C05476=1016.184,128.856,379.831,166.835,54.880,160.081
C05477=1016.188,129.105,379.813,166.839,54.870,160.080
C05478=1016.193,129.355,379.795,166.841,54.860,160.079
C05479=1016.197,129.605,379.776,166.845,54.850,160.077
C05480=1016.202,129.853,379.757,166.848,54.840,160.076
C05481=1016.207,130.103,379.739,166.851,54.831,160.075
C05482=1016.211,130.352,379.720,166.854,54.820,160.073
C05483=1016.216,130.601,379.702,166.858,54.811,160.072
C05484=1016.220,130.851,379.683,166.860,54.801,160.071
C05485=1016.225,131.099,379.664,166.863,54.791,160.069
C05486=1016.231,131.349,379.645,166.867,54.781,160.068
C05487=1016.235,131.598,379.626,166.869,54.771,160.067
C05488=1016.240,131.848,379.608,166.873,54.761,160.066
C05489=1016.244,132.097,379.589,166.876,54.751,160.065
C05490=1016.249,132.346,379.570,166.879,54.741,160.063
C05491=1016.254,132.596,379.552,166.882,54.731,160.062
C05492=1016.258,132.845,379.533,166.886,54.721,160.061
C05493=1016.263,133.094,379.514,166.888,54.712,160.059
C05494=1016.267,133.343,379.495,166.891,54.701,160.058
C05495=1016.272,133.592,379.477,166.895,54.692,160.057
C05496=1016.277,133.841,379.458,166.898,54.681,160.055
C05497=1016.282,134.091,379.439,166.901,54.672,160.054
C05498=1016.287,134.340,379.420,166.904,54.662,160.053
C05499=1016.291,134.590,379.401,166.908,54.652,160.052
C05500=1016.296,134.839,379.382,166.910,54.642,160.050
C05501=1016.301,135.088,379.364,166.914,54.632,160.049
C05502=1016.305,135.337,379.345,166.917,54.622,160.048
C05503=1016.310,135.586,379.326,166.921,54.612,160.046
C05504=1016.314,135.835,379.307,166.923,54.602,160.045
C05505=1016.320,136.085,379.288,166.927,54.592,160.044
C05506=1016.324,136.334,379.269,166.930,54.582,160.043
C05507=1016.329,136.583,379.250,166.932,54.572,160.041
C05508=1016.333,136.833,379.231,166.936,54.563,160.040
C05509=1016.338,137.082,379.212,166.939,54.552,160.039
C05510=1016.342,137.331,379.194,166.943,54.542,160.037
C05511=1016.348,137.581,379.174,166.946,54.533,160.036
C05512=1016.352,137.830,379.155,166.949,54.523,160.035
C05513=1016.357,138.079,379.137,166.952,54.512,160.034
C05514=1016.361,138.328,379.117,166.955,54.503,160.032
C05515=1016.366,138.609,379.095,166.959,54.492,160.031
C05516=1016.372,138.890,379.074,166.963,54.481,160.030
C05517=1016.377,139.171,379.053,166.966,54.470,160.028
C05518=1016.382,139.452,379.031,166.970,54.458,160.027
C05519=1016.387,139.702,379.011,166.974,54.449,160.026
C05520=1016.392,139.951,378.993,166.977,54.439,160.024
C05521=1016.396,140.200,378.973,166.980,54.429,160.023
C05522=1016.400,140.449,378.954,166.983,54.419,160.022
C05523=1016.406,140.699,378.935,166.986,54.409,160.020
C05524=1016.410,140.948,378.915,166.989,54.400,160.019
C05525=1016.415,141.197,378.896,166.993,54.390,160.018
C05526=1016.420,141.446,378.878,166.996,54.379,160.017
C05527=1016.424,141.695,378.858,167.000,54.370,160.016
C05528=1016.429,141.945,378.838,167.002,54.360,160.014
C05529=1016.434,142.194,378.819,167.006,54.350,160.013
C05530=1016.438,142.443,378.800,167.010,54.340,160.012
C05531=1016.442,142.692,378.781,167.013,54.330,160.010
C05532=1016.448,142.942,378.762,167.015,54.320,160.009
C05533=1016.452,143.191,378.742,167.019,54.311,160.008
C05534=1016.457,143.440,378.723,167.023,54.301,160.007
C05535=1016.462,143.689,378.704,167.026,54.290,160.005
C05536=1016.467,143.938,378.684,167.029,54.281,160.004
C05537=1016.471,144.187,378.665,167.032,54.271,160.003
C05538=1016.476,144.436,378.646,167.036,54.261,160.001
C05539=1016.481,144.686,378.626,167.040,54.251,160.000
C05540=1016.485,144.935,378.607,167.043,54.241,159.999
C05541=1016.490,145.184,378.588,167.045,54.231,159.998
C05542=1016.495,145.434,378.569,167.049,54.222,159.997
C05543=1016.500,145.683,378.549,167.053,54.212,159.995
C05544=1016.504,145.932,378.530,167.056,54.202,159.994
C05545=1016.509,146.182,378.510,167.059,54.192,159.993
C05546=1016.514,146.430,378.491,167.062,54.182,159.991
C05547=1016.518,146.680,378.472,167.066,54.173,159.990
C05548=1016.523,146.928,378.451,167.070,54.163,159.989
C05549=1016.528,147.178,378.431,167.072,54.153,159.988
C05550=1016.532,147.427,378.412,167.076,54.143,159.987
C05551=1016.537,147.676,378.392,167.080,54.133,159.985
C05552=1016.542,147.926,378.373,167.083,54.124,159.984
C05553=1016.546,148.175,378.353,167.086,54.114,159.983
C05554=1016.552,148.424,378.334,167.089,54.104,159.982
C05555=1016.556,148.673,378.315,167.093,54.094,159.980
C05556=1016.560,148.922,378.295,167.097,54.084,159.979
C05557=1016.566,149.171,378.274,167.100,54.075,159.978
C05558=1016.570,149.420,378.255,167.103,54.065,159.977
C05559=1016.574,149.669,378.236,167.107,54.055,159.975
C05560=1016.579,149.919,378.216,167.110,54.045,159.974
C05561=1016.584,150.168,378.196,167.113,54.035,159.973
C05562=1016.589,150.418,378.176,167.117,54.026,159.972
C05563=1016.593,150.666,378.156,167.120,54.016,159.971
C05564=1016.598,150.915,378.137,167.124,54.006,159.969
C05565=1016.602,151.165,378.117,167.128,53.996,159.968
C05566=1016.607,151.414,378.097,167.130,53.986,159.967
C05567=1016.612,151.663,378.077,167.134,53.977,159.966
C05568=1016.616,151.912,378.057,167.138,53.967,159.964
C05569=1016.621,152.161,378.038,167.141,53.957,159.963
C05570=1016.626,152.411,378.018,167.145,53.947,159.962
C05571=1016.630,152.659,377.998,167.148,53.938,159.961
C05572=1016.635,152.909,377.978,167.152,53.928,159.960
C05573=1016.640,153.158,377.959,167.155,53.918,159.958
C05574=1016.645,153.407,377.938,167.159,53.908,159.957
C05575=1016.649,153.656,377.919,167.162,53.898,159.956
C05576=1016.654,153.906,377.899,167.165,53.889,159.954
C05577=1016.659,154.155,377.879,167.169,53.879,159.953
C05578=1016.663,154.404,377.859,167.172,53.869,159.952
C05579=1016.668,154.685,377.835,167.177,53.858,159.951
C05580=1016.674,154.966,377.814,167.181,53.847,159.950
C05581=1016.679,155.247,377.791,167.184,53.837,159.948
C05582=1016.685,155.528,377.769,167.188,53.825,159.947
C05583=1016.689,155.778,377.748,167.192,53.815,159.945
C05584=1016.693,156.026,377.728,167.196,53.806,159.944
C05585=1016.698,156.276,377.708,167.199,53.796,159.943
C05586=1016.703,156.524,377.688,167.203,53.786,159.942
C05587=1016.708,156.774,377.668,167.206,53.777,159.941
C05588=1016.713,157.022,377.648,167.210,53.767,159.940
C05589=1016.718,157.272,377.628,167.213,53.757,159.938
C05590=1016.722,157.521,377.608,167.217,53.747,159.937
C05591=1016.727,157.770,377.588,167.221,53.738,159.936
C05592=1016.731,158.019,377.567,167.224,53.727,159.935
C05593=1016.736,158.269,377.547,167.227,53.718,159.933
C05594=1016.741,158.517,377.527,167.231,53.708,159.932
C05595=1016.746,158.767,377.507,167.235,53.699,159.931
C05596=1016.750,159.016,377.487,167.238,53.689,159.930
C05597=1016.754,159.265,377.465,167.241,53.680,159.929
C05598=1016.759,159.514,377.445,167.245,53.670,159.928
C05599=1016.763,159.764,377.425,167.249,53.660,159.926
C05600=1016.768,160.012,377.405,167.253,53.651,159.925
C05601=1016.772,160.261,377.383,167.256,53.642,159.924
C05602=1016.777,160.511,377.363,167.260,53.632,159.923
C05603=1016.781,160.759,377.342,167.264,53.623,159.922
C05604=1016.785,161.009,377.322,167.268,53.613,159.921
C05605=1016.790,161.258,377.302,167.270,53.603,159.919
C05606=1016.795,161.507,377.280,167.274,53.594,159.918
C05607=1016.799,161.756,377.260,167.278,53.584,159.917
C05608=1016.804,162.005,377.239,167.282,53.575,159.916
C05609=1016.808,162.255,377.218,167.285,53.566,159.915
C05610=1016.813,162.504,377.198,167.288,53.556,159.913
C05611=1016.817,162.753,377.177,167.292,53.546,159.912
C05612=1016.822,163.001,377.157,167.297,53.537,159.911
C05613=1016.826,163.251,377.136,167.299,53.527,159.910
C05614=1016.832,163.500,377.115,167.303,53.518,159.909
C05615=1016.836,163.749,377.095,167.307,53.508,159.908
C05616=1016.840,163.998,377.073,167.311,53.498,159.906
C05617=1016.845,164.247,377.053,167.315,53.489,159.905
C05618=1016.849,164.496,377.032,167.317,53.479,159.904
C05619=1016.855,164.745,377.012,167.321,53.470,159.903
C05620=1016.858,164.994,376.991,167.325,53.460,159.902
C05621=1016.863,165.244,376.970,167.329,53.451,159.901
C05622=1016.868,165.493,376.950,167.333,53.441,159.900
C05623=1016.872,165.742,376.929,167.337,53.431,159.898
C05624=1016.877,165.991,376.908,167.340,53.422,159.897
C05625=1016.882,166.240,376.887,167.343,53.412,159.896
C05626=1016.885,166.489,376.867,167.348,53.403,159.895
C05627=1016.891,166.738,376.846,167.352,53.394,159.894
C05628=1016.895,166.988,376.825,167.355,53.384,159.892
C05629=1016.900,167.236,376.805,167.359,53.374,159.891
C05630=1016.904,167.486,376.783,167.362,53.365,159.890
C05631=1016.909,167.735,376.762,167.366,53.355,159.889
C05632=1016.914,167.984,376.742,167.370,53.346,159.888
C05633=1016.918,168.233,376.721,167.374,53.336,159.887
C05634=1016.923,168.482,376.700,167.378,53.327,159.886
C05635=1016.928,168.731,376.679,167.381,53.317,159.884
C05636=1016.932,168.979,376.658,167.386,53.307,159.883
C05637=1016.937,169.229,376.637,167.390,53.298,159.882
C05638=1016.942,169.478,376.616,167.393,53.288,159.881
C05639=1016.947,169.727,376.596,167.396,53.279,159.880
C05640=1016.951,169.976,376.575,167.400,53.269,159.878
C05641=1016.956,170.225,376.554,167.404,53.260,159.877
C05642=1016.961,170.474,376.533,167.408,53.250,159.876
C05643=1016.966,170.755,376.509,167.412,53.239,159.875
C05644=1016.971,171.036,376.485,167.417,53.228,159.874
C05645=1016.977,171.317,376.462,167.421,53.218,159.872
C05646=1016.983,171.597,376.438,167.426,53.207,159.871
C05647=1016.986,171.846,376.417,167.429,53.197,159.870
C05648=1016.992,172.095,376.397,167.433,53.187,159.869
C05649=1016.996,172.345,376.376,167.438,53.178,159.868
C05650=1017.001,172.594,376.354,167.441,53.168,159.866
C05651=1017.006,172.843,376.334,167.445,53.159,159.865
C05652=1017.011,173.092,376.312,167.449,53.149,159.864
C05653=1017.015,173.340,376.292,167.453,53.140,159.863
C05654=1017.020,173.590,376.271,167.457,53.130,159.862
C05655=1017.024,173.839,376.250,167.461,53.120,159.861
C05656=1017.030,174.088,376.228,167.465,53.110,159.859
C05657=1017.035,174.337,376.207,167.469,53.101,159.858
C05658=1017.039,174.587,376.186,167.473,53.092,159.857
C05659=1017.044,174.836,376.165,167.477,53.082,159.856
C05660=1017.049,175.084,376.144,167.481,53.073,159.855
C05661=1017.054,175.333,376.123,167.484,53.063,159.854
C05662=1017.058,175.582,376.102,167.489,53.053,159.853
C05663=1017.063,175.831,376.080,167.492,53.043,159.851
C05664=1017.068,176.080,376.060,167.496,53.034,159.850
C05665=1017.073,176.330,376.039,167.500,53.024,159.849
C05666=1017.078,176.579,376.018,167.504,53.015,159.848
C05667=1017.083,176.828,375.996,167.508,53.006,159.847
C05668=1017.088,177.077,375.975,167.512,52.996,159.846
C05669=1017.093,177.326,375.954,167.516,52.986,159.845
C05670=1017.098,177.575,375.933,167.520,52.976,159.843
C05671=1017.102,177.825,375.912,167.524,52.967,159.842
C05672=1017.108,178.073,375.890,167.528,52.957,159.841
C05673=1017.112,178.323,375.869,167.532,52.948,159.840
C05674=1017.117,178.571,375.849,167.536,52.938,159.839
C05675=1017.122,178.820,375.827,167.540,52.929,159.838
C05676=1017.126,179.069,375.806,167.544,52.919,159.837
C05677=1017.132,179.318,375.785,167.548,52.910,159.835
C05678=1017.136,179.567,375.764,167.553,52.899,159.834
C05679=1017.141,179.816,375.742,167.557,52.890,159.833
C05680=1017.146,180.065,375.721,167.561,52.881,159.832
C05681=1017.151,180.315,375.700,167.565,52.871,159.831
C05682=1017.156,180.563,375.679,167.569,52.862,159.830
C05683=1017.161,180.812,375.658,167.573,52.852,159.829
C05684=1017.166,181.062,375.635,167.577,52.843,159.828
C05685=1017.172,181.311,375.615,167.581,52.833,159.826
C05686=1017.176,181.560,375.593,167.585,52.823,159.825
C05687=1017.181,181.809,375.572,167.590,52.813,159.824
C05688=1017.186,182.058,375.550,167.594,52.804,159.823
C05689=1017.191,182.307,375.528,167.597,52.795,159.822
C05690=1017.195,182.556,375.506,167.601,52.786,159.821
C05691=1017.199,182.806,375.484,167.605,52.777,159.820
C05692=1017.204,183.054,375.463,167.610,52.767,159.819
C05693=1017.209,183.303,375.441,167.614,52.758,159.818
C05694=1017.213,183.552,375.418,167.618,52.749,159.817
C05695=1017.218,183.801,375.396,167.622,52.739,159.815
C05696=1017.223,184.050,375.375,167.626,52.730,159.814
C05697=1017.227,184.299,375.353,167.630,52.721,159.813
C05698=1017.232,184.548,375.330,167.635,52.711,159.812
C05699=1017.236,184.797,375.308,167.639,52.702,159.811
C05700=1017.241,185.045,375.286,167.643,52.693,159.810
C05701=1017.245,185.295,375.265,167.647,52.684,159.809
C05702=1017.250,185.544,375.243,167.651,52.675,159.808
C05703=1017.255,185.794,375.221,167.655,52.665,159.807
C05704=1017.260,186.042,375.199,167.659,52.656,159.806
C05705=1017.264,186.292,375.176,167.664,52.646,159.805
C05706=1017.269,186.540,375.154,167.668,52.637,159.804
C05707=1017.275,186.820,375.129,167.673,52.627,159.803
C05708=1017.280,187.101,375.104,167.677,52.616,159.801
C05709=1017.285,187.381,375.080,167.682,52.606,159.800
C05710=1017.290,187.662,375.055,167.687,52.596,159.799
C05711=1017.294,187.910,375.033,167.691,52.586,159.798
C05712=1017.300,188.160,375.011,167.695,52.577,159.797
C05713=1017.304,188.409,374.988,167.699,52.568,159.796
C05714=1017.309,188.658,374.966,167.703,52.558,159.795
C05715=1017.314,188.906,374.944,167.708,52.549,159.794
C05716=1017.319,189.155,374.922,167.712,52.540,159.792
C05717=1017.323,189.404,374.900,167.716,52.531,159.791
C05718=1017.328,189.654,374.877,167.721,52.521,159.791
C05719=1017.333,189.902,374.855,167.726,52.512,159.789
C05720=1017.337,190.152,374.833,167.730,52.503,159.788
C05721=1017.342,190.400,374.811,167.734,52.494,159.787
C05722=1017.347,190.649,374.789,167.738,52.484,159.786
C05723=1017.352,190.899,374.767,167.742,52.475,159.785
C05724=1017.357,191.147,374.744,167.746,52.465,159.784
C05725=1017.361,191.396,374.722,167.751,52.456,159.783
C05726=1017.366,191.645,374.700,167.755,52.447,159.782
C05727=1017.371,191.895,374.677,167.759,52.438,159.781
C05728=1017.376,192.143,374.655,167.765,52.429,159.780
C05729=1017.381,192.392,374.633,167.769,52.419,159.779
C05730=1017.386,192.640,374.611,167.773,52.410,159.778
C05731=1017.390,192.890,374.588,167.777,52.400,159.777
C05732=1017.395,193.139,374.566,167.781,52.391,159.776
C05733=1017.400,193.387,374.544,167.786,52.382,159.775
C05734=1017.405,193.637,374.521,167.790,52.373,159.774
C05735=1017.410,193.886,374.499,167.795,52.364,159.773
C05736=1017.415,194.135,374.477,167.799,52.354,159.772
C05737=1017.419,194.383,374.454,167.804,52.345,159.771
C05738=1017.424,194.633,374.432,167.808,52.335,159.769
C05739=1017.429,194.882,374.410,167.812,52.326,159.768
C05740=1017.434,195.130,374.387,167.816,52.317,159.767
C05741=1017.439,195.380,374.364,167.822,52.308,159.766
C05742=1017.444,195.628,374.343,167.826,52.299,159.765
C05743=1017.450,195.877,374.320,167.830,52.289,159.764
C05744=1017.454,196.126,374.297,167.834,52.280,159.763
C05745=1017.459,196.375,374.275,167.839,52.271,159.762
C05746=1017.464,196.624,374.252,167.844,52.262,159.761
C05747=1017.468,196.873,374.230,167.848,52.253,159.760
C05748=1017.474,197.121,374.207,167.852,52.243,159.759
C05749=1017.479,197.371,374.185,167.857,52.234,159.758
C05750=1017.483,197.620,374.163,167.862,52.224,159.757
C05751=1017.489,197.869,374.140,167.866,52.215,159.756
C05752=1017.494,198.118,374.118,167.871,52.206,159.755
C05753=1017.499,198.367,374.095,167.875,52.197,159.754
C05754=1017.503,198.616,374.072,167.880,52.188,159.753
C05755=1017.509,198.864,374.050,167.885,52.178,159.752
C05756=1017.514,199.114,374.028,167.889,52.169,159.751
C05757=1017.518,199.362,374.004,167.893,52.160,159.750
C05758=1017.523,199.612,373.982,167.899,52.151,159.749
C05759=1017.528,199.860,373.959,167.903,52.142,159.748
C05760=1017.533,200.109,373.936,167.907,52.133,159.747
C05761=1017.537,200.358,373.913,167.912,52.124,159.746
C05762=1017.543,200.607,373.890,167.916,52.114,159.745
C05763=1017.547,200.856,373.867,167.920,52.105,159.744
C05764=1017.552,201.104,373.844,167.926,52.096,159.743
C05765=1017.557,201.354,373.822,167.930,52.087,159.742
C05766=1017.562,201.602,373.798,167.935,52.078,159.741
C05767=1017.567,201.852,373.775,167.939,52.069,159.740
C05768=1017.572,202.100,373.752,167.943,52.060,159.739
C05769=1017.577,202.349,373.729,167.949,52.051,159.738
C05770=1017.600,203.593,373.613,168.432,52.137,159.849
C05771=1017.606,203.828,373.591,168.436,52.129,159.848
C05772=1017.612,204.063,373.567,168.440,52.122,159.847
C05773=1017.618,204.298,373.544,168.443,52.114,159.846
C05774=1017.623,204.534,373.521,168.447,52.107,159.845
C05775=1017.629,204.769,373.498,168.450,52.099,159.844
C05776=1017.634,205.003,373.474,168.454,52.091,159.844
C05777=1017.640,205.238,373.451,168.458,52.084,159.843
C05778=1017.645,205.473,373.428,168.462,52.076,159.842
C05779=1017.651,205.722,373.402,168.466,52.068,159.841
C05780=1017.657,205.970,373.378,168.470,52.061,159.840
C05781=1017.663,206.219,373.353,168.474,52.053,159.839
C05782=1017.669,206.468,373.328,168.477,52.045,159.838
C05783=1017.674,206.716,373.303,168.481,52.037,159.837
C05784=1017.680,206.966,373.279,168.485,52.030,159.836
C05785=1017.686,207.214,373.254,168.490,52.021,159.835
C05786=1017.692,207.463,373.229,168.494,52.013,159.834
C05787=1017.698,207.712,373.204,168.498,52.006,159.834
C05788=1017.703,207.960,373.179,168.501,51.998,159.833
C05789=1017.709,208.209,373.154,168.505,51.990,159.832
C05790=1017.716,208.458,373.129,168.509,51.983,159.831
C05791=1017.721,208.706,373.104,168.513,51.975,159.830
C05792=1017.727,208.955,373.079,168.517,51.967,159.829
C05793=1017.732,209.204,373.054,168.521,51.960,159.828
C05794=1017.738,209.452,373.029,168.525,51.951,159.827
C05795=1017.744,209.701,373.004,168.530,51.944,159.826
C05796=1017.750,209.950,372.978,168.533,51.936,159.825
C05797=1017.756,210.198,372.954,168.537,51.929,159.825
C05798=1017.762,210.447,372.929,168.541,51.921,159.824
C05799=1017.767,210.696,372.903,168.545,51.913,159.823
C05800=1017.773,210.944,372.878,168.549,51.905,159.822
C05801=1017.779,211.193,372.853,168.553,51.898,159.821
C05802=1017.785,211.442,372.828,168.557,51.890,159.820
C05803=1017.790,211.690,372.802,168.561,51.883,159.819
C05804=1017.796,211.939,372.777,168.565,51.876,159.818
C05805=1017.802,212.187,372.752,168.569,51.868,159.817
C05806=1017.808,212.436,372.726,168.573,51.860,159.817
C05807=1017.813,212.685,372.701,168.577,51.853,159.816
C05808=1017.819,212.934,372.676,168.581,51.845,159.815
C05809=1017.825,213.182,372.651,168.585,51.838,159.814
C05810=1017.831,213.431,372.625,168.589,51.830,159.813
C05811=1017.836,213.679,372.600,168.593,51.823,159.812
C05812=1017.843,213.928,372.574,168.597,51.816,159.811
C05813=1017.849,214.177,372.549,168.601,51.808,159.810
C05814=1017.854,214.426,372.523,168.605,51.800,159.810
C05815=1017.860,214.674,372.499,168.609,51.793,159.809
C05816=1017.866,214.923,372.474,168.613,51.786,159.808
C05817=1017.871,215.172,372.448,168.617,51.778,159.807
C05818=1017.878,215.421,372.422,168.621,51.771,159.806
C05819=1017.884,215.669,372.397,168.625,51.763,159.806
C05820=1017.889,215.917,372.372,168.630,51.756,159.805
C05821=1017.895,216.166,372.346,168.633,51.748,159.804
C05822=1017.901,216.415,372.321,168.636,51.741,159.803
C05823=1017.907,216.663,372.295,168.641,51.734,159.802
C05824=1017.913,216.912,372.270,168.645,51.727,159.801
C05825=1017.919,217.161,372.244,168.648,51.719,159.800
C05826=1017.925,217.410,372.219,168.653,51.712,159.799
C05827=1017.931,217.658,372.194,168.657,51.704,159.799
C05828=1017.937,217.906,372.168,168.661,51.697,159.798
C05829=1017.943,218.155,372.142,168.665,51.690,159.797
C05830=1017.949,218.403,372.116,168.669,51.683,159.796
C05831=1017.959,218.817,372.074,168.675,51.671,159.795
C05832=1017.966,219.179,372.036,168.681,51.660,159.794
C05833=1017.975,219.540,371.998,168.687,51.650,159.793
C05834=1017.983,219.901,371.961,168.693,51.640,159.792
C05835=1017.992,220.263,371.923,168.699,51.629,159.790
C05836=1017.998,220.512,371.897,168.704,51.622,159.790
C05837=1018.003,220.760,371.872,168.708,51.615,159.789
C05838=1018.009,221.009,371.846,168.712,51.608,159.788
C05839=1018.015,221.257,371.820,168.716,51.600,159.787
C05840=1018.021,221.506,371.794,168.719,51.594,159.786
C05841=1018.026,221.755,371.768,168.723,51.586,159.786
C05842=1018.033,222.003,371.742,168.728,51.580,159.785
C05843=1018.038,222.252,371.716,168.732,51.573,159.784
C05844=1018.044,222.500,371.691,168.736,51.565,159.783
C05845=1018.050,222.749,371.664,168.741,51.558,159.783
C05846=1018.056,222.997,371.639,168.744,51.551,159.782
C05847=1018.062,223.246,371.613,168.748,51.544,159.781
C05848=1018.068,223.495,371.587,168.753,51.537,159.780
C05849=1018.074,223.743,371.561,168.757,51.530,159.780
C05850=1018.080,223.992,371.535,168.761,51.523,159.779
C05851=1018.086,224.240,371.509,168.765,51.516,159.778
C05852=1018.091,224.489,371.483,168.769,51.510,159.777
C05853=1018.097,224.738,371.457,168.773,51.502,159.777
C05854=1018.103,224.986,371.431,168.777,51.495,159.776
C05855=1018.109,225.235,371.405,168.781,51.488,159.775
C05856=1018.115,225.483,371.379,168.786,51.482,159.774
C05857=1018.121,225.732,371.353,168.789,51.475,159.774
C05858=1018.127,225.980,371.327,168.793,51.467,159.773
C05859=1018.133,226.229,371.301,168.798,51.461,159.772
C05860=1018.138,226.478,371.275,168.802,51.454,159.771
C05861=1018.145,226.726,371.249,168.806,51.447,159.771
C05862=1018.151,226.974,371.222,168.810,51.440,159.770
C05863=1018.156,227.223,371.196,168.814,51.433,159.769
C05864=1018.162,227.471,371.169,168.819,51.427,159.769
C05865=1018.168,227.720,371.142,168.822,51.420,159.768
C05866=1018.174,227.969,371.117,168.827,51.413,159.767
C05867=1018.180,228.218,371.090,168.831,51.406,159.766
C05868=1018.186,228.466,371.064,168.836,51.400,159.766
C05869=1018.191,228.715,371.038,168.839,51.393,159.765
C05870=1018.197,228.963,371.011,168.843,51.386,159.764
C05871=1018.203,229.212,370.985,168.848,51.379,159.764
C05872=1018.209,229.460,370.958,168.851,51.373,159.763
C05873=1018.215,229.709,370.933,168.856,51.366,159.762
C05874=1018.221,229.957,370.906,168.860,51.359,159.762
C05875=1018.227,230.205,370.879,168.865,51.353,159.761
C05876=1018.233,230.454,370.852,168.868,51.347,159.760
C05877=1018.239,230.703,370.826,168.873,51.339,159.759
C05878=1018.244,230.951,370.799,168.877,51.333,159.759
C05879=1018.250,231.199,370.772,168.881,51.327,159.758
C05880=1018.256,231.448,370.746,168.885,51.320,159.757
C05881=1018.262,231.697,370.720,168.890,51.313,159.757
C05882=1018.267,231.945,370.693,168.893,51.307,159.756
C05883=1018.274,232.194,370.666,168.898,51.300,159.755
C05884=1018.279,232.443,370.639,168.902,51.293,159.755
C05885=1018.285,232.691,370.613,168.906,51.287,159.754
C05886=1018.291,232.939,370.586,168.911,51.281,159.754
C05887=1018.297,233.188,370.559,168.914,51.275,159.753
C05888=1018.302,233.416,370.535,168.919,51.268,159.752
C05889=1018.308,233.644,370.510,168.922,51.262,159.752
C05890=1018.313,233.872,370.486,168.926,51.256,159.751
C05891=1018.318,234.101,370.461,168.930,51.250,159.750
C05892=1018.324,234.329,370.437,168.934,51.244,159.750
C05893=1018.330,234.558,370.412,168.937,51.238,159.749
C05894=1018.334,234.786,370.387,168.941,51.233,159.749
C05895=1018.341,235.014,370.363,168.945,51.226,159.748
C05896=1018.346,235.262,370.337,168.950,51.220,159.747
C05897=1018.353,235.511,370.310,168.954,51.213,159.747
C05898=1018.358,235.760,370.283,168.958,51.207,159.746
C05899=1018.365,236.007,370.256,168.963,51.201,159.746
C05900=1018.370,236.256,370.229,168.966,51.195,159.745
C05901=1018.377,236.505,370.202,168.971,51.188,159.744
C05902=1018.382,236.753,370.175,168.976,51.182,159.744
C05903=1018.387,237.002,370.148,168.979,51.176,159.743
C05904=1018.393,237.250,370.121,168.984,51.169,159.743
C05905=1018.400,237.499,370.094,168.988,51.162,159.742
C05906=1018.406,237.747,370.067,168.992,51.156,159.741
C05907=1018.412,237.995,370.040,168.997,51.150,159.741
C05908=1018.418,238.244,370.013,169.000,51.144,159.740
C05909=1018.424,238.493,369.987,169.005,51.138,159.739
C05910=1018.429,238.741,369.960,169.010,51.131,159.739
C05911=1018.436,238.990,369.932,169.013,51.125,159.738
C05912=1018.442,239.238,369.906,169.018,51.118,159.738
C05913=1018.447,239.487,369.878,169.022,51.112,159.737
C05914=1018.454,239.735,369.851,169.026,51.106,159.736
C05915=1018.459,239.983,369.824,169.030,51.100,159.736
C05916=1018.465,240.231,369.796,169.035,51.094,159.735
C05917=1018.471,240.481,369.769,169.039,51.088,159.735
C05918=1018.477,240.729,369.742,169.043,51.081,159.734
C05919=1018.483,240.978,369.714,169.047,51.075,159.733
C05920=1018.489,241.226,369.687,169.052,51.070,159.733
C05921=1018.495,241.474,369.660,169.056,51.063,159.732
C05922=1018.500,241.723,369.632,169.061,51.057,159.732
C05923=1018.506,241.971,369.605,169.064,51.051,159.731
C05924=1018.513,242.220,369.578,169.069,51.045,159.731
C05925=1018.518,242.468,369.550,169.074,51.039,159.730
C05926=1018.524,242.716,369.523,169.078,51.033,159.729
C05927=1018.531,242.965,369.496,169.083,51.027,159.729
C05928=1018.536,243.213,369.468,169.086,51.021,159.728
C05929=1018.542,243.462,369.441,169.091,51.015,159.728
C05930=1018.548,243.710,369.413,169.095,51.009,159.727
C05931=1018.553,243.958,369.385,169.099,51.003,159.727
C05932=1018.559,244.207,369.358,169.104,50.997,159.726
C05933=1018.565,244.455,369.330,169.107,50.991,159.726
C05934=1018.571,244.704,369.302,169.113,50.985,159.725
C05935=1018.576,244.952,369.275,169.117,50.980,159.725
C05936=1018.582,245.201,369.247,169.121,50.973,159.724
C05937=1018.588,245.449,369.219,169.125,50.968,159.724
C05938=1018.594,245.697,369.191,169.130,50.961,159.723
C05939=1018.600,245.945,369.163,169.134,50.956,159.723
C05940=1018.606,246.195,369.136,169.138,50.950,159.722
C05941=1018.611,246.443,369.108,169.143,50.944,159.722
C05942=1018.617,246.691,369.080,169.147,50.939,159.721
C05943=1018.623,246.939,369.052,169.152,50.932,159.720
C05944=1018.629,247.188,369.024,169.156,50.927,159.720
C05945=1018.635,247.436,368.997,169.160,50.920,159.719
C05946=1018.641,247.685,368.969,169.164,50.915,159.719
C05947=1018.646,247.933,368.941,169.169,50.910,159.718
C05948=1018.652,248.158,368.915,169.173,50.904,159.718
C05949=1018.657,248.383,368.891,169.177,50.899,159.718
C05950=1018.663,248.608,368.865,169.181,50.893,159.717
C05951=1018.668,248.833,368.840,169.185,50.888,159.717
C05952=1018.674,249.058,368.815,169.189,50.883,159.716
C05953=1018.679,249.283,368.790,169.192,50.878,159.716
C05954=1018.684,249.507,368.765,169.196,50.873,159.715
C05955=1018.689,249.733,368.738,169.201,50.867,159.715
C05956=1018.696,249.981,368.711,169.205,50.862,159.714
C05957=1018.701,250.229,368.683,169.210,50.856,159.714
C05958=1018.708,250.478,368.655,169.214,50.851,159.714
C05959=1018.714,250.726,368.627,169.218,50.844,159.713
C05960=1018.719,250.974,368.599,169.223,50.839,159.712
C05961=1018.726,251.223,368.571,169.228,50.833,159.712
C05962=1018.731,251.471,368.543,169.232,50.828,159.712
C05963=1018.737,251.720,368.515,169.236,50.822,159.711
C05964=1018.744,251.968,368.487,169.240,50.816,159.711
C05965=1018.749,252.216,368.459,169.245,50.811,159.710
C05966=1018.755,252.465,368.431,169.250,50.805,159.710
C05967=1018.762,252.713,368.403,169.254,50.799,159.709
C05968=1018.767,252.961,368.375,169.259,50.794,159.709
C05969=1018.773,253.210,368.347,169.263,50.788,159.708
C05970=1018.780,253.459,368.319,169.267,50.783,159.708
C05971=1018.786,253.706,368.290,169.272,50.777,159.707
C05972=1018.792,253.954,368.262,169.276,50.771,159.707
C05973=1018.798,254.203,368.234,169.281,50.765,159.706
C05974=1018.804,254.452,368.206,169.285,50.760,159.706
C05975=1018.810,254.700,368.178,169.290,50.754,159.706
C05976=1018.816,254.948,368.150,169.294,50.749,159.705
C05977=1018.823,255.197,368.121,169.298,50.744,159.705
C05978=1018.829,255.445,368.093,169.303,50.738,159.704
C05979=1018.835,255.693,368.065,169.307,50.732,159.704
C05980=1018.840,255.942,368.037,169.313,50.727,159.703
C05981=1018.847,256.190,368.009,169.317,50.721,159.703
C05982=1018.853,256.438,367.980,169.322,50.716,159.703
C05983=1018.859,256.687,367.952,169.326,50.710,159.702
C05984=1018.865,256.935,367.925,169.330,50.705,159.702
C05985=1018.872,257.183,367.896,169.335,50.699,159.701
C05986=1018.878,257.432,367.867,169.339,50.694,159.701
C05987=1018.884,257.680,367.839,169.344,50.688,159.700
C05988=1018.891,257.928,367.810,169.348,50.683,159.700
C05989=1018.896,258.177,367.782,169.352,50.677,159.699
C05990=1018.903,258.425,367.755,169.358,50.672,159.699
C05991=1018.909,258.673,367.726,169.362,50.667,159.699
C05992=1018.915,258.922,367.697,169.367,50.661,159.698
C05993=1018.922,259.170,367.669,169.371,50.656,159.698
C05994=1018.928,259.418,367.641,169.376,50.650,159.697
C05995=1018.934,259.667,367.612,169.380,50.645,159.697
C05996=1018.941,259.915,367.584,169.385,50.639,159.697
C05997=1018.946,260.162,367.555,169.390,50.634,159.696
C05998=1018.952,260.411,367.527,169.394,50.629,159.696
C05999=1018.958,260.659,367.498,169.398,50.624,159.695
C06000=1018.965,260.907,367.469,169.404,50.618,159.695
C06001=1018.971,261.156,367.440,169.408,50.613,159.695
C06002=1018.976,261.404,367.411,169.412,50.608,159.694
C06003=1018.982,261.653,367.382,169.417,50.603,159.694
C06004=1018.988,261.901,367.353,169.422,50.597,159.694
C06005=1018.995,262.149,367.324,169.426,50.593,159.693
C06006=1019.000,262.397,367.296,169.431,50.587,159.693
C06007=1019.007,262.645,367.267,169.436,50.582,159.693
C06008=1019.012,262.870,367.241,169.440,50.578,159.692
C06009=1019.018,263.094,367.215,169.444,50.573,159.692
C06010=1019.023,263.318,367.188,169.448,50.569,159.692
C06011=1019.028,263.542,367.163,169.453,50.564,159.691
C06012=1019.034,263.766,367.137,169.457,50.558,159.691
C06013=1019.040,263.990,367.110,169.460,50.554,159.691
C06014=1019.045,264.214,367.084,169.465,50.549,159.690
C06015=1019.051,264.439,367.058,169.469,50.545,159.690
C06016=1019.057,264.687,367.029,169.474,50.540,159.690
C06017=1019.063,264.936,367.000,169.478,50.535,159.689
C06018=1019.069,265.184,366.971,169.483,50.530,159.689
C06019=1019.076,265.432,366.942,169.488,50.525,159.689
C06020=1019.082,265.680,366.913,169.492,50.520,159.688
C06021=1019.087,265.928,366.883,169.496,50.515,159.688
C06022=1019.094,266.176,366.854,169.502,50.510,159.688
C06023=1019.100,266.425,366.825,169.506,50.505,159.687
C06024=1019.106,266.673,366.796,169.511,50.500,159.687
C06025=1019.112,266.921,366.766,169.516,50.495,159.687
C06026=1019.118,267.169,366.737,169.520,50.490,159.686
C06027=1019.124,267.417,366.708,169.525,50.485,159.686
C06028=1019.130,267.666,366.679,169.530,50.480,159.686
C06029=1019.136,267.914,366.650,169.535,50.475,159.686
C06030=1019.142,268.162,366.621,169.539,50.470,159.685
C06031=1019.149,268.410,366.591,169.543,50.465,159.685
C06032=1019.155,268.658,366.562,169.549,50.460,159.685
C06033=1019.161,268.906,366.532,169.553,50.455,159.685
C06034=1019.167,269.154,366.503,169.558,50.451,159.684
C06035=1019.173,269.403,366.474,169.563,50.445,159.684
C06036=1019.179,269.651,366.445,169.568,50.440,159.684
C06037=1019.186,269.899,366.414,169.572,50.436,159.683
C06038=1019.192,270.147,366.385,169.577,50.431,159.683
C06039=1019.197,270.396,366.356,169.582,50.426,159.683
C06040=1019.204,270.643,366.326,169.587,50.421,159.683
C06041=1019.209,270.892,366.296,169.591,50.417,159.682
C06042=1019.216,271.140,366.267,169.596,50.412,159.682
C06043=1019.222,271.387,366.237,169.601,50.407,159.682
C06044=1019.228,271.636,366.207,169.606,50.402,159.682
C06045=1019.235,271.885,366.178,169.610,50.398,159.681
C06046=1019.240,272.132,366.148,169.615,50.393,159.681
C06047=1019.247,272.381,366.119,169.620,50.388,159.681
C06048=1019.252,272.629,366.089,169.625,50.383,159.681
C06049=1019.259,272.877,366.059,169.629,50.379,159.680
C06050=1019.265,273.126,366.030,169.634,50.374,159.680
C06051=1019.271,273.373,366.000,169.639,50.369,159.680
C06052=1019.277,273.622,365.970,169.644,50.364,159.679
C06053=1019.284,273.869,365.941,169.648,50.360,159.679
C06054=1019.290,274.118,365.911,169.653,50.355,159.679
C06055=1019.296,274.366,365.881,169.659,50.351,159.679
C06056=1019.302,274.614,365.851,169.663,50.346,159.679
C06057=1019.308,274.862,365.821,169.668,50.341,159.678
C06058=1019.315,275.110,365.791,169.672,50.337,159.678
C06059=1019.321,275.358,365.762,169.678,50.332,159.678
C06060=1019.327,275.606,365.731,169.683,50.328,159.678
C06061=1019.334,275.855,365.702,169.687,50.323,159.678
C06062=1019.339,276.103,365.671,169.692,50.318,159.677
C06063=1019.346,276.350,365.642,169.697,50.313,159.677
C06064=1019.351,276.599,365.612,169.702,50.309,159.677
C06065=1019.359,276.847,365.582,169.707,50.305,159.677
C06066=1019.364,277.095,365.552,169.711,50.300,159.676
C06067=1019.370,277.343,365.521,169.717,50.295,159.676
C06068=1019.376,277.570,365.494,169.720,50.291,159.676
C06069=1019.382,277.796,365.467,169.725,50.287,159.676
C06070=1019.387,278.022,365.439,169.730,50.283,159.676
C06071=1019.393,278.249,365.411,169.734,50.279,159.676
C06072=1019.398,278.475,365.383,169.739,50.275,159.675
C06073=1019.404,278.701,365.356,169.744,50.271,159.675
C06074=1019.410,278.928,365.329,169.747,50.267,159.675
C06075=1019.415,279.154,365.301,169.752,50.263,159.675
C06076=1019.422,279.403,365.270,169.757,50.259,159.675
C06077=1019.428,279.650,365.240,169.761,50.254,159.675
C06078=1019.435,279.899,365.209,169.767,50.250,159.675
C06079=1019.440,280.147,365.180,169.772,50.245,159.674
C06080=1019.446,280.395,365.150,169.777,50.241,159.674
C06081=1019.452,280.643,365.119,169.781,50.237,159.674
C06082=1019.459,280.891,365.089,169.787,50.232,159.674
C06083=1019.465,281.139,365.058,169.792,50.228,159.674
C06084=1019.471,281.387,365.028,169.797,50.224,159.674
C06085=1019.477,281.636,364.997,169.801,50.220,159.673
C06086=1019.484,281.883,364.967,169.806,50.215,159.673
C06087=1019.491,282.131,364.936,169.812,50.211,159.673
C06088=1019.497,282.379,364.906,169.816,50.206,159.673
C06089=1019.502,282.627,364.875,169.821,50.202,159.673
C06090=1019.509,282.875,364.845,169.826,50.198,159.673
C06091=1019.515,283.123,364.815,169.832,50.193,159.673
C06092=1019.522,283.371,364.784,169.837,50.189,159.672
C06093=1019.528,283.620,364.753,169.842,50.185,159.672
C06094=1019.534,283.868,364.723,169.846,50.180,159.672
C06095=1019.541,284.115,364.692,169.852,50.176,159.672
C06096=1019.547,284.363,364.662,169.857,50.172,159.672
C06097=1019.554,284.612,364.631,169.861,50.168,159.672
C06098=1019.560,284.859,364.601,169.866,50.164,159.672
C06099=1019.566,285.107,364.569,169.871,50.160,159.672
C06100=1019.572,285.355,364.539,169.877,50.155,159.672
C06101=1019.578,285.604,364.508,169.882,50.151,159.671
C06102=1019.585,285.851,364.477,169.887,50.147,159.671
C06103=1019.591,286.099,364.447,169.891,50.143,159.671
C06104=1019.597,286.348,364.416,169.896,50.139,159.671
C06105=1019.604,286.595,364.385,169.902,50.134,159.671
C06106=1019.610,286.844,364.354,169.907,50.130,159.671
C06107=1019.616,287.091,364.323,169.912,50.126,159.671
C06108=1019.623,287.339,364.292,169.917,50.123,159.671
C06109=1019.629,287.587,364.261,169.923,50.118,159.671
C06110=1019.635,287.835,364.230,169.928,50.114,159.671
C06111=1019.642,288.083,364.199,169.933,50.110,159.671
C06112=1019.648,288.332,364.168,169.938,50.106,159.670
C06113=1019.654,288.579,364.137,169.943,50.102,159.670
C06114=1019.661,288.827,364.107,169.948,50.098,159.670
C06115=1019.667,289.075,364.075,169.953,50.094,159.670
C06116=1019.673,289.323,364.045,169.958,50.090,159.670
C06117=1019.680,289.571,364.013,169.963,50.086,159.670
C06118=1019.687,289.819,363.982,169.968,50.082,159.670
C06119=1019.693,290.067,363.952,169.974,50.078,159.670
C06120=1019.699,290.315,363.920,169.979,50.074,159.670
C06121=1019.705,290.563,363.888,169.984,50.070,159.670
C06122=1019.711,290.811,363.858,169.989,50.066,159.670
C06123=1019.718,291.058,363.826,169.994,50.062,159.670
C06124=1019.725,291.306,363.795,170.000,50.058,159.670
C06125=1019.731,291.554,363.763,170.005,50.054,159.670
C06126=1019.737,291.802,363.733,170.010,50.050,159.670
C06127=1019.743,292.050,363.701,170.015,50.046,159.670
C06128=1019.750,292.283,363.672,170.020,50.043,159.670
C06129=1019.755,292.516,363.642,170.025,50.039,159.670
C06130=1019.762,292.748,363.613,170.030,50.036,159.670
C06131=1019.767,292.981,363.583,170.035,50.032,159.670
C06132=1019.774,293.213,363.554,170.039,50.028,159.669
C06133=1019.779,293.446,363.524,170.044,50.025,159.670
C06134=1019.785,293.678,363.495,170.050,50.022,159.670
C06135=1019.791,293.910,363.464,170.054,50.018,159.670
C06136=1019.797,294.158,363.433,170.060,50.014,159.670
C06137=1019.803,294.406,363.401,170.065,50.010,159.670
C06138=1019.810,294.654,363.369,170.070,50.007,159.670
C06139=1019.816,294.902,363.337,170.075,50.003,159.670
C06140=1019.822,295.150,363.306,170.080,50.000,159.670
C06141=1019.828,295.398,363.274,170.086,49.996,159.670
C06142=1019.834,295.645,363.242,170.091,49.992,159.670
C06143=1019.841,295.893,363.210,170.096,49.988,159.670
C06144=1019.847,296.142,363.178,170.102,49.985,159.670
C06145=1019.854,296.389,363.147,170.106,49.981,159.670
C06146=1019.860,296.638,363.115,170.112,49.978,159.670
C06147=1019.866,296.884,363.083,170.118,49.974,159.670
C06148=1019.872,297.132,363.051,170.123,49.970,159.670
C06149=1019.878,297.381,363.019,170.128,49.967,159.670
C06150=1019.885,297.628,362.987,170.133,49.963,159.670
C06151=1019.891,297.876,362.955,170.138,49.960,159.670
C06152=1019.898,298.124,362.923,170.144,49.956,159.670
C06153=1019.904,298.372,362.890,170.150,49.952,159.670
C06154=1019.911,298.620,362.859,170.155,49.949,159.670
C06155=1019.917,298.868,362.827,170.160,49.946,159.670
C06156=1019.923,299.115,362.794,170.165,49.942,159.671
C06157=1019.930,299.363,362.763,170.170,49.938,159.670
C06158=1019.936,299.611,362.731,170.177,49.935,159.671
C06159=1019.943,299.859,362.699,170.182,49.931,159.671
C06160=1019.949,300.107,362.667,170.187,49.928,159.671
C06161=1019.956,300.354,362.634,170.192,49.924,159.671
C06162=1019.962,300.602,362.602,170.197,49.921,159.671
C06163=1019.968,300.850,362.570,170.204,49.917,159.671
C06164=1019.975,301.098,362.538,170.209,49.914,159.671
C06165=1019.981,301.346,362.505,170.214,49.911,159.671
C06166=1019.988,301.593,362.474,170.219,49.907,159.671
C06167=1019.994,301.841,362.441,170.225,49.903,159.671
C06168=1020.001,302.089,362.409,170.231,49.900,159.671
C06169=1020.007,302.337,362.377,170.236,49.896,159.672
C06170=1020.014,302.585,362.344,170.241,49.893,159.672
C06171=1020.021,302.833,362.313,170.247,49.890,159.672
C06172=1020.027,303.080,362.280,170.252,49.887,159.672
C06173=1020.034,303.328,362.248,170.258,49.883,159.672
C06174=1020.040,303.576,362.216,170.264,49.880,159.672
C06175=1020.047,303.823,362.183,170.268,49.876,159.672
C06176=1020.054,304.071,362.151,170.274,49.872,159.672
C06177=1020.060,304.320,362.118,170.280,49.869,159.672
C06178=1020.067,304.567,362.086,170.285,49.866,159.672
C06179=1020.073,304.814,362.054,170.291,49.862,159.673
C06180=1020.080,305.062,362.021,170.296,49.859,159.673
C06181=1020.087,305.309,361.989,170.302,49.855,159.673
C06182=1020.093,305.558,361.956,170.308,49.853,159.673
C06183=1020.100,305.806,361.924,170.313,49.849,159.673
C06184=1020.107,306.053,361.891,170.318,49.846,159.673
C06185=1020.113,306.301,361.859,170.325,49.843,159.674
C06186=1020.121,306.549,361.826,170.330,49.839,159.674
C06187=1020.127,306.796,361.793,170.335,49.836,159.674
C06188=1020.133,307.038,361.762,170.341,49.833,159.674
C06189=1020.140,307.279,361.730,170.346,49.829,159.674
C06190=1020.147,307.521,361.699,170.353,49.826,159.674
C06191=1020.154,307.761,361.667,170.358,49.823,159.674
C06192=1020.160,308.003,361.635,170.363,49.820,159.675
C06193=1020.166,308.245,361.604,170.368,49.817,159.675
C06194=1020.173,308.485,361.572,170.374,49.813,159.675
C06195=1020.180,308.727,361.540,170.379,49.811,159.675
C06196=1020.186,308.975,361.507,170.385,49.807,159.675
C06197=1020.193,309.223,361.474,170.391,49.804,159.675
C06198=1020.200,309.470,361.442,170.396,49.800,159.675
C06199=1020.207,309.718,361.409,170.402,49.798,159.676
C06200=1020.214,309.966,361.377,170.408,49.794,159.676
C06201=1020.220,310.213,361.343,170.414,49.792,159.676
C06202=1020.226,310.461,361.310,170.419,49.788,159.676
C06203=1020.234,310.708,361.276,170.425,49.786,159.677
C06204=1020.240,310.956,361.243,170.430,49.782,159.677
C06205=1020.247,311.203,361.210,170.437,49.779,159.677
C06206=1020.253,311.452,361.176,170.442,49.776,159.677
C06207=1020.259,311.699,361.144,170.448,49.774,159.677
C06208=1020.266,311.946,361.110,170.453,49.771,159.678
C06209=1020.272,312.194,361.077,170.459,49.768,159.678
C06210=1020.278,312.442,361.043,170.465,49.765,159.678
C06211=1020.286,312.689,361.009,170.471,49.761,159.678
C06212=1020.292,312.937,360.976,170.476,49.759,159.679
C06213=1020.299,313.185,360.943,170.482,49.756,159.679
C06214=1020.305,313.433,360.909,170.488,49.753,159.679
C06215=1020.312,313.680,360.875,170.494,49.750,159.679
C06216=1020.318,313.928,360.843,170.500,49.747,159.680
C06217=1020.325,314.176,360.809,170.505,49.745,159.680
C06218=1020.331,314.423,360.775,170.511,49.741,159.680
C06219=1020.338,314.671,360.742,170.517,49.738,159.681
C06220=1020.345,314.918,360.708,170.523,49.736,159.681
C06221=1020.352,315.166,360.674,170.529,49.733,159.681
C06222=1020.358,315.413,360.640,170.534,49.731,159.681
C06223=1020.365,315.661,360.607,170.541,49.727,159.682
C06224=1020.371,315.908,360.574,170.546,49.724,159.682
C06225=1020.378,316.156,360.540,170.552,49.722,159.682
C06226=1020.385,316.404,360.505,170.558,49.719,159.682
C06227=1020.391,316.652,360.473,170.564,49.716,159.683
C06228=1020.398,316.899,360.439,170.570,49.713,159.683
C06229=1020.405,317.146,360.405,170.575,49.711,159.683
C06230=1020.411,317.394,360.371,170.581,49.708,159.684
C06231=1020.419,317.642,360.337,170.587,49.705,159.684
C06232=1020.425,317.889,360.304,170.593,49.702,159.684
C06233=1020.432,318.136,360.270,170.599,49.699,159.684
C06234=1020.439,318.384,360.235,170.605,49.696,159.685
C06235=1020.446,318.633,360.202,170.611,49.694,159.685
C06236=1020.452,318.880,360.169,170.617,49.691,159.685
C06237=1020.460,319.127,360.135,170.622,49.688,159.686
C06238=1020.466,319.375,360.101,170.629,49.686,159.686
C06239=1020.473,319.622,360.067,170.635,49.683,159.686
C06240=1020.480,319.870,360.033,170.641,49.681,159.687
C06241=1020.487,320.118,360.000,170.647,49.678,159.687
C06242=1020.493,320.366,359.965,170.653,49.675,159.688
C06243=1020.501,320.613,359.931,170.659,49.673,159.688
C06244=1020.508,320.860,359.897,170.665,49.670,159.688
C06245=1020.514,321.108,359.863,170.671,49.667,159.689
C06246=1020.521,321.355,359.829,170.677,49.665,159.689
C06247=1020.528,321.603,359.795,170.683,49.662,159.689
C06248=1020.535,321.847,359.762,170.689,49.660,159.690
C06249=1020.542,322.091,359.728,170.695,49.657,159.690
C06250=1020.549,322.335,359.694,170.701,49.654,159.690
C06251=1020.555,322.579,359.661,170.707,49.651,159.691
C06252=1020.563,322.822,359.627,170.713,49.649,159.691
C06253=1020.569,323.066,359.593,170.719,49.647,159.691
C06254=1020.577,323.310,359.560,170.725,49.644,159.692
C06255=1020.584,323.554,359.526,170.731,49.641,159.692
C06256=1020.590,323.802,359.492,170.737,49.639,159.693
C06257=1020.598,324.049,359.458,170.744,49.636,159.693
C06258=1020.605,324.297,359.424,170.750,49.634,159.693
C06259=1020.612,324.544,359.390,170.756,49.632,159.694
C06260=1020.619,324.792,359.355,170.762,49.629,159.694
C06261=1020.626,325.039,359.321,170.768,49.626,159.694
C06262=1020.633,325.286,359.286,170.774,49.624,159.695
C06263=1020.640,325.535,359.252,170.781,49.621,159.695
C06264=1020.648,325.783,359.218,170.787,49.619,159.696
C06265=1020.655,326.030,359.183,170.794,49.616,159.696
C06266=1020.662,326.278,359.149,170.799,49.614,159.696
C06267=1020.669,326.525,359.114,170.805,49.612,159.697
C06268=1020.677,326.772,359.080,170.812,49.609,159.697
C06269=1020.683,327.020,359.045,170.818,49.607,159.698
C06270=1020.690,327.267,359.010,170.825,49.604,159.698
C06271=1020.697,327.515,358.975,170.831,49.602,159.699
C06272=1020.704,327.762,358.940,170.837,49.600,159.699
C06273=1020.711,328.010,358.906,170.844,49.597,159.700
C06274=1020.717,328.257,358.871,170.849,49.595,159.700
C06275=1020.725,328.504,358.836,170.855,49.593,159.700
C06276=1020.732,328.752,358.801,170.862,49.591,159.701
C06277=1020.739,328.999,358.766,170.868,49.589,159.702
C06278=1020.746,329.247,358.731,170.874,49.586,159.702
C06279=1020.753,329.494,358.696,170.881,49.584,159.702
C06280=1020.760,329.742,358.662,170.887,49.582,159.703
C06281=1020.767,329.989,358.627,170.894,49.579,159.703
C06282=1020.774,330.237,358.591,170.900,49.577,159.704
C06283=1020.781,330.484,358.556,170.906,49.575,159.704
C06284=1020.788,330.732,358.521,170.913,49.572,159.705
C06285=1020.795,330.979,358.486,170.919,49.570,159.705
C06286=1020.802,331.226,358.451,170.926,49.568,159.706
C06287=1020.810,331.474,358.415,170.932,49.566,159.706
C06288=1020.817,331.721,358.380,170.939,49.564,159.707
C06289=1020.824,331.968,358.345,170.945,49.562,159.707
C06290=1020.831,332.216,358.310,170.951,49.560,159.708
C06291=1020.839,332.463,358.275,170.958,49.558,159.708
C06292=1020.845,332.711,358.240,170.964,49.556,159.709
C06293=1020.853,332.959,358.205,170.971,49.553,159.709
C06294=1020.860,333.206,358.169,170.977,49.551,159.710
C06295=1020.867,333.453,358.134,170.984,49.549,159.711
C06296=1020.874,333.701,358.098,170.990,49.547,159.711
C06297=1020.881,333.948,358.062,170.997,49.546,159.712
C06298=1020.888,334.195,358.027,171.004,49.543,159.712
C06299=1020.895,334.443,357.992,171.010,49.541,159.713
C06300=1020.902,334.690,357.956,171.017,49.539,159.713
C06301=1020.909,334.937,357.921,171.023,49.537,159.714
C06302=1020.917,335.185,357.884,171.030,49.535,159.715
C06303=1020.923,335.432,357.849,171.036,49.533,159.715
C06304=1020.931,335.680,357.813,171.043,49.531,159.716
C06305=1020.938,335.927,357.778,171.049,49.529,159.716
C06306=1020.945,336.174,357.742,171.056,49.528,159.717
C06307=1020.952,336.422,357.707,171.063,49.526,159.717
C06308=1020.959,336.663,357.671,171.069,49.524,159.718
C06309=1020.967,336.905,357.637,171.076,49.522,159.719
C06310=1020.974,337.146,357.602,171.082,49.520,159.719
C06311=1020.981,337.388,357.567,171.088,49.518,159.720
C06312=1020.988,337.630,357.532,171.095,49.516,159.720
C06313=1020.995,337.872,357.496,171.101,49.514,159.721
C06314=1021.002,338.114,357.462,171.108,49.513,159.721
C06315=1021.009,338.355,357.426,171.115,49.511,159.722
C06316=1021.016,338.602,357.390,171.121,49.509,159.723
C06317=1021.024,338.850,357.355,171.128,49.507,159.723
C06318=1021.031,339.097,357.319,171.135,49.506,159.724
C06319=1021.039,339.344,357.283,171.142,49.503,159.725
C06320=1021.046,339.591,357.247,171.148,49.502,159.725
C06321=1021.053,339.838,357.211,171.155,49.500,159.726
C06322=1021.061,340.086,357.174,171.161,49.498,159.726
C06323=1021.068,340.333,357.138,171.169,49.497,159.727
C06324=1021.075,340.580,357.102,171.175,49.495,159.728
C06325=1021.083,340.828,357.066,171.182,49.493,159.728
C06326=1021.090,341.075,357.029,171.189,49.492,159.729
C06327=1021.097,341.322,356.993,171.196,49.489,159.730
C06328=1021.104,341.570,356.957,171.202,49.488,159.730
C06329=1021.112,341.817,356.920,171.209,49.486,159.731
C06330=1021.119,342.064,356.885,171.217,49.485,159.732
C06331=1021.126,342.312,356.848,171.223,49.483,159.733
C06332=1021.134,342.558,356.811,171.230,49.481,159.733
C06333=1021.142,342.806,356.775,171.237,49.480,159.734
C06334=1021.149,343.053,356.739,171.244,49.478,159.735
C06335=1021.156,343.300,356.702,171.250,49.477,159.735
C06336=1021.164,343.547,356.665,171.258,49.475,159.736
C06337=1021.171,343.795,356.628,171.265,49.473,159.737
C06338=1021.178,344.042,356.592,171.272,49.472,159.738
C06339=1021.186,344.288,356.555,171.279,49.470,159.738
C06340=1021.193,344.536,356.519,171.285,49.469,159.739
C06341=1021.200,344.784,356.482,171.293,49.467,159.740
C06342=1021.208,345.030,356.446,171.299,49.466,159.740
C06343=1021.215,345.278,356.409,171.307,49.464,159.741
C06344=1021.223,345.525,356.372,171.314,49.462,159.742
C06345=1021.231,345.772,356.336,171.320,49.461,159.743
C06346=1021.238,346.020,356.298,171.328,49.459,159.743
C06347=1021.246,346.267,356.262,171.335,49.458,159.744
C06348=1021.254,346.514,356.225,171.341,49.456,159.745
C06349=1021.261,346.762,356.188,171.349,49.455,159.746
C06350=1021.268,347.008,356.152,171.357,49.454,159.747
C06351=1021.275,347.255,356.114,171.363,49.452,159.747
C06352=1021.283,347.502,356.078,171.370,49.451,159.748
C06353=1021.290,347.749,356.040,171.377,49.449,159.749
C06354=1021.298,347.996,356.003,171.385,49.448,159.750
C06355=1021.305,348.244,355.967,171.392,49.446,159.750
C06356=1021.313,348.491,355.930,171.398,49.445,159.751
C06357=1021.320,348.738,355.892,171.406,49.444,159.752
C06358=1021.329,348.986,355.855,171.413,49.442,159.753
C06359=1021.336,349.233,355.817,171.420,49.441,159.753
C06360=1021.343,349.480,355.780,171.428,49.440,159.754
C06361=1021.351,349.727,355.743,171.435,49.438,159.755
C06362=1021.359,349.974,355.705,171.442,49.438,159.756
C06363=1021.367,350.221,355.668,171.449,49.436,159.757
C06364=1021.374,350.468,355.631,171.457,49.435,159.758
C06365=1021.381,350.715,355.593,171.464,49.433,159.758
C06366=1021.389,350.962,355.556,171.471,49.432,159.759
C06367=1021.396,351.209,355.519,171.478,49.431,159.760
C06368=1021.404,351.449,355.482,171.485,49.430,159.761
C06369=1021.411,351.690,355.446,171.493,49.428,159.762
C06370=1021.419,351.930,355.409,171.500,49.427,159.763
C06371=1021.427,352.170,355.372,171.507,49.426,159.764
C06372=1021.434,352.410,355.337,171.514,49.425,159.764
C06373=1021.441,352.650,355.300,171.521,49.424,159.765
C06374=1021.449,352.890,355.263,171.529,49.422,159.766
C06375=1021.457,353.130,355.226,171.535,49.422,159.767
C06376=1021.465,353.377,355.189,171.543,49.421,159.768
C06377=1021.472,353.624,355.152,171.551,49.420,159.769
C06378=1021.480,353.872,355.114,171.558,49.418,159.770
C06379=1021.488,354.118,355.076,171.566,49.417,159.771
C06380=1021.495,354.365,355.039,171.573,49.416,159.771
C06381=1021.503,354.613,355.000,171.580,49.415,159.772
C06382=1021.511,354.860,354.963,171.588,49.414,159.773
C06383=1021.518,355.106,354.925,171.596,49.413,159.774
C06384=1021.527,355.354,354.887,171.603,49.412,159.775
C06385=1021.534,355.600,354.849,171.610,49.411,159.776
C06386=1021.542,355.847,354.811,171.618,49.410,159.777
C06387=1021.550,356.095,354.773,171.626,49.409,159.778
C06388=1021.557,356.341,354.735,171.634,49.408,159.779
C06389=1021.566,356.589,354.697,171.641,49.407,159.780
C06390=1021.573,356.835,354.659,171.648,49.406,159.781
C06391=1021.582,357.082,354.620,171.656,49.405,159.782
C06392=1021.589,357.329,354.582,171.664,49.404,159.783
C06393=1021.597,357.577,354.544,171.671,49.403,159.784
C06394=1021.605,357.823,354.506,171.679,49.402,159.785
C06395=1021.613,358.071,354.467,171.687,49.401,159.786
C06396=1021.621,358.317,354.430,171.695,49.400,159.787
C06397=1021.629,358.564,354.391,171.702,49.399,159.788
C06398=1021.637,358.811,354.353,171.710,49.398,159.789
C06399=1021.645,359.058,354.314,171.717,49.397,159.790
C06400=1021.652,359.304,354.276,171.725,49.397,159.791
C06401=1021.661,359.551,354.237,171.733,49.396,159.792
C06402=1021.669,359.799,354.199,171.741,49.395,159.793
C06403=1021.676,360.045,354.161,171.749,49.394,159.794
C06404=1021.684,360.292,354.122,171.757,49.393,159.795
C06405=1021.692,360.539,354.084,171.764,49.392,159.796
C06406=1021.700,360.786,354.045,171.773,49.392,159.797
C06407=1021.708,361.034,354.006,171.780,49.391,159.798
C06408=1021.715,361.280,353.967,171.787,49.390,159.799
C06409=1021.724,361.527,353.928,171.795,49.389,159.800
C06410=1021.732,361.774,353.890,171.803,49.389,159.801
C06411=1021.740,362.020,353.851,171.811,49.388,159.802
C06412=1021.748,362.267,353.812,171.819,49.387,159.803
C06413=1021.756,362.514,353.774,171.827,49.387,159.804
C06414=1021.764,362.761,353.734,171.835,49.386,159.805
C06415=1021.771,363.008,353.695,171.843,49.385,159.806
C06416=1021.780,363.254,353.656,171.851,49.385,159.808
C06417=1021.788,363.502,353.618,171.859,49.384,159.809
C06418=1021.796,363.748,353.578,171.867,49.383,159.810
C06419=1021.804,363.995,353.540,171.875,49.383,159.811
C06420=1021.811,364.242,353.500,171.883,49.382,159.812
C06421=1021.820,364.489,353.461,171.891,49.382,159.813
C06422=1021.828,364.735,353.422,171.899,49.381,159.814
C06423=1021.837,364.982,353.383,171.907,49.380,159.815
C06424=1021.845,365.229,353.344,171.915,49.380,159.816
C06425=1021.853,365.476,353.305,171.924,49.379,159.818
C06426=1021.861,365.723,353.265,171.933,49.379,159.819
C06427=1021.869,365.969,353.226,171.941,49.378,159.820
C06428=1021.877,366.213,353.187,171.949,49.378,159.821
C06429=1021.885,366.457,353.149,171.957,49.377,159.822
C06430=1021.893,366.700,353.110,171.965,49.377,159.823
C06431=1021.902,366.944,353.071,171.973,49.376,159.825
C06432=1021.910,367.187,353.032,171.981,49.376,159.826
C06433=1021.919,367.431,352.994,171.989,49.375,159.827
C06434=1021.927,367.675,352.954,171.997,49.375,159.828
C06435=1021.935,367.918,352.916,172.006,49.374,159.829
C06436=1021.943,368.165,352.876,172.014,49.374,159.830
C06437=1021.951,368.412,352.837,172.022,49.373,159.832
C06438=1021.959,368.658,352.797,172.030,49.374,159.833
C06439=1021.968,368.904,352.757,172.038,49.373,159.834
C06440=1021.976,369.152,352.716,172.048,49.372,159.835
C06441=1021.984,369.399,352.677,172.056,49.372,159.836
C06442=1021.992,369.646,352.637,172.064,49.372,159.838
C06443=1022.001,369.891,352.597,172.072,49.372,159.839
C06444=1022.009,370.138,352.557,172.081,49.372,159.840
C06445=1022.017,370.385,352.518,172.089,49.371,159.841
C06446=1022.025,370.631,352.477,172.098,49.371,159.843
C06447=1022.034,370.879,352.438,172.106,49.370,159.844
C06448=1022.042,371.125,352.397,172.115,49.371,159.845
C06449=1022.051,371.371,352.358,172.123,49.370,159.847
C06450=1022.059,371.618,352.317,172.132,49.370,159.848
C06451=1022.068,371.865,352.277,172.141,49.369,159.849
C06452=1022.076,372.111,352.237,172.149,49.370,159.851
C06453=1022.084,372.358,352.197,172.157,49.369,159.852
C06454=1022.092,372.604,352.157,172.167,49.369,159.853
C06455=1022.102,372.851,352.116,172.175,49.369,159.854
C06456=1022.109,373.098,352.076,172.183,49.368,159.856
C06457=1022.118,373.344,352.036,172.192,49.369,159.857
C06458=1022.127,373.591,351.995,172.201,49.368,159.858
C06459=1022.135,373.837,351.956,172.210,49.369,159.860
C06460=1022.144,374.084,351.915,172.218,49.368,159.861
C06461=1022.153,374.330,351.875,172.227,49.368,159.862
C06462=1022.161,374.577,351.834,172.236,49.368,159.864
C06463=1022.170,374.823,351.794,172.245,49.368,159.865
C06464=1022.178,375.071,351.754,172.254,49.368,159.867
C06465=1022.187,375.317,351.714,172.262,49.368,159.868
C06466=1022.196,375.564,351.673,172.272,49.368,159.869
C06467=1022.204,375.810,351.632,172.280,49.368,159.871
C06468=1022.213,376.057,351.591,172.288,49.368,159.872
C06469=1022.222,376.303,351.551,172.298,49.368,159.873
C06470=1022.230,376.550,351.510,172.306,49.368,159.875
C06471=1022.239,376.795,351.469,172.316,49.368,159.876
C06472=1022.247,377.042,351.428,172.324,49.368,159.878
C06473=1022.256,377.288,351.388,172.334,49.368,159.879
C06474=1022.265,377.535,351.346,172.342,49.368,159.880
C06475=1022.274,377.782,351.305,172.351,49.368,159.882
C06476=1022.282,378.028,351.265,172.361,49.368,159.883
C06477=1022.291,378.274,351.223,172.369,49.368,159.885
C06478=1022.299,378.521,351.182,172.379,49.369,159.886
C06479=1022.308,378.767,351.141,172.387,49.369,159.888
C06480=1022.317,379.014,351.100,172.397,49.368,159.889
C06481=1022.326,379.260,351.059,172.406,49.369,159.891
C06482=1022.334,379.506,351.018,172.415,49.369,159.892
C06483=1022.343,379.753,350.976,172.424,49.370,159.894
C06484=1022.352,380.000,350.935,172.433,49.369,159.895
C06485=1022.361,380.246,350.893,172.442,49.370,159.897
C06486=1022.370,380.491,350.853,172.452,49.370,159.898
C06487=1022.378,380.738,350.812,172.461,49.371,159.900
C06488=1022.387,380.982,350.771,172.470,49.370,159.901
C06489=1022.396,381.226,350.729,172.479,49.371,159.903
C06490=1022.404,381.470,350.689,172.488,49.371,159.904
C06491=1022.413,381.713,350.647,172.498,49.371,159.906
C06492=1022.423,381.957,350.606,172.507,49.372,159.907
C06493=1022.431,382.201,350.565,172.517,49.372,159.909
C06494=1022.440,382.445,350.524,172.525,49.372,159.910
C06495=1022.449,382.689,350.483,172.535,49.373,159.912
C06496=1022.458,382.935,350.441,172.544,49.373,159.914
C06497=1022.467,383.181,350.400,172.554,49.373,159.915
C06498=1022.476,383.428,350.358,172.563,49.373,159.917
C06499=1022.485,383.674,350.317,172.573,49.374,159.918
C06500=1022.494,383.920,350.275,172.582,49.374,159.920
C06501=1022.504,384.166,350.233,172.592,49.375,159.922
C06502=1022.512,384.412,350.191,172.602,49.375,159.923
C06503=1022.521,384.659,350.149,172.611,49.376,159.925
C06504=1022.530,384.905,350.108,172.620,49.376,159.926
C06505=1022.540,385.151,350.066,172.630,49.377,159.928
C06506=1022.549,385.397,350.024,172.640,49.377,159.930
C06507=1022.559,385.644,349.982,172.650,49.377,159.931
C06508=1022.568,385.890,349.940,172.659,49.378,159.933
C06509=1022.577,386.136,349.898,172.669,49.379,159.935
C06510=1022.586,386.382,349.856,172.679,49.379,159.936
C06511=1022.594,386.628,349.813,172.689,49.380,159.938
C06512=1022.604,386.876,349.771,172.698,49.380,159.940
C06513=1022.613,387.121,349.728,172.708,49.381,159.942
C06514=1022.622,387.367,349.686,172.718,49.381,159.943
C06515=1022.631,387.613,349.644,172.727,49.382,159.945
C06516=1022.641,387.860,349.602,172.738,49.383,159.947
C06517=1022.650,388.106,349.559,172.747,49.383,159.948
C06518=1022.659,388.352,349.517,172.758,49.384,159.950
C06519=1022.668,388.599,349.474,172.767,49.384,159.952
C06520=1022.678,388.844,349.432,172.778,49.385,159.954
C06521=1022.687,389.090,349.389,172.788,49.386,159.956
C06522=1022.697,389.337,349.346,172.797,49.387,159.957
C06523=1022.706,389.582,349.304,172.807,49.388,159.959
C06524=1022.715,389.828,349.261,172.817,49.389,159.961
C06525=1022.724,390.075,349.218,172.827,49.389,159.962
C06526=1022.734,390.321,349.176,172.837,49.390,159.964
C06527=1022.743,390.567,349.132,172.847,49.391,159.966
C06528=1022.752,390.813,349.090,172.858,49.392,159.968
C06529=1022.762,391.059,349.046,172.867,49.392,159.970
C06530=1022.771,391.305,349.004,172.878,49.393,159.971
C06531=1022.780,391.551,348.960,172.888,49.394,159.973
C06532=1022.791,391.818,348.914,172.899,49.395,159.975
C06533=1022.801,392.086,348.867,172.911,49.396,159.977
C06534=1022.812,392.353,348.820,172.922,49.397,159.980
C06535=1022.823,392.621,348.773,172.932,49.398,159.981
C06536=1022.832,392.866,348.731,172.944,49.398,159.983
C06537=1022.841,393.113,348.687,172.954,49.399,159.985
C06538=1022.851,393.359,348.644,172.964,49.401,159.987
C06539=1022.860,393.605,348.600,172.975,49.402,159.989
C06540=1022.870,393.851,348.557,172.985,49.402,159.991
C06541=1022.879,394.097,348.513,172.995,49.403,159.993
C06542=1022.889,394.342,348.470,173.006,49.405,159.995
C06543=1022.898,394.589,348.427,173.017,49.405,159.997
C06544=1022.908,394.835,348.383,173.027,49.406,159.999
C06545=1022.918,395.081,348.340,173.038,49.408,160.001
C06546=1022.927,395.326,348.296,173.048,49.409,160.003
C06547=1022.937,395.572,348.252,173.059,49.410,160.005
C06548=1022.949,395.872,348.199,173.072,49.411,160.007
C06549=1022.961,396.172,348.146,173.085,49.413,160.010
C06550=1022.972,396.471,348.093,173.098,49.414,160.012
C06551=1022.984,396.770,348.039,173.111,49.415,160.014
C06552=1022.994,397.016,347.995,173.121,49.416,160.016
C06553=1023.004,397.262,347.952,173.133,49.417,160.018
C06554=1023.013,397.507,347.907,173.143,49.419,160.020
C06555=1023.024,397.753,347.864,173.154,49.420,160.022
C06556=1023.033,397.999,347.819,173.165,49.421,160.024
C06557=1023.043,398.245,347.776,173.176,49.422,160.026
C06558=1023.053,398.491,347.731,173.186,49.424,160.029
C06559=1023.063,398.736,347.688,173.198,49.425,160.031
C06560=1023.073,398.983,347.642,173.209,49.426,160.033
C06561=1023.083,399.229,347.598,173.220,49.427,160.035
C06562=1023.093,399.474,347.554,173.231,49.429,160.037
C06563=1023.103,399.720,347.510,173.242,49.430,160.039
C06564=1023.112,399.966,347.465,173.253,49.431,160.041
C06565=1023.122,400.212,347.422,173.264,49.433,160.043
C06566=1023.132,400.457,347.377,173.275,49.434,160.045
C06567=1023.142,400.703,347.332,173.287,49.435,160.048
C06568=1023.153,400.948,347.287,173.298,49.437,160.050
C06569=1023.162,401.195,347.243,173.309,49.438,160.052
C06570=1023.172,401.440,347.198,173.320,49.440,160.054
C06571=1023.182,401.686,347.153,173.332,49.441,160.056
C06572=1023.192,401.932,347.108,173.343,49.442,160.058
C06573=1023.202,402.177,347.064,173.354,49.444,160.061
C06574=1023.213,402.423,347.019,173.366,49.446,160.063
C06575=1023.223,402.669,346.974,173.377,49.448,160.065
C06576=1023.233,402.914,346.929,173.388,49.449,160.067
C06577=1023.243,403.160,346.883,173.400,49.450,160.070
C06578=1023.253,403.405,346.839,173.411,49.452,160.072
C06579=1023.263,403.652,346.793,173.423,49.453,160.074
C06580=1023.273,403.897,346.749,173.435,49.455,160.076
C06581=1023.283,404.143,346.703,173.447,49.457,160.079
C06582=1023.294,404.388,346.658,173.457,49.458,160.081
C06583=1023.304,404.634,346.613,173.469,49.460,160.083
C06584=1023.314,404.879,346.568,173.481,49.461,160.086
C06585=1023.324,405.125,346.523,173.493,49.463,160.088
C06586=1023.335,405.371,346.477,173.504,49.465,160.090
C06587=1023.345,405.616,346.432,173.516,49.467,160.093
C06588=1023.355,405.862,346.386,173.528,49.468,160.095
C06589=1023.367,406.107,346.341,173.540,49.470,160.097
C06590=1023.376,406.353,346.296,173.552,49.472,160.100
C06591=1023.387,406.598,346.250,173.564,49.473,160.102
C06592=1023.398,406.844,346.204,173.576,49.475,160.104
C06593=1023.408,407.090,346.159,173.588,49.477,160.107
C06594=1023.419,407.336,346.113,173.600,49.478,160.109
C06595=1023.429,407.581,346.067,173.612,49.480,160.112
C06596=1023.439,407.826,346.021,173.624,49.482,160.114
C06597=1023.451,408.071,345.976,173.636,49.484,160.116
C06598=1023.461,408.317,345.930,173.648,49.486,160.119
C06599=1023.472,408.563,345.884,173.660,49.487,160.121
C06600=1023.482,408.808,345.838,173.672,49.489,160.124
C06601=1023.493,409.054,345.792,173.684,49.491,160.126
C06602=1023.504,409.299,345.747,173.696,49.493,160.129
C06603=1023.514,409.545,345.701,173.709,49.495,160.131
C06604=1023.525,409.791,345.655,173.721,49.497,160.134
C06605=1023.536,410.036,345.608,173.733,49.499,160.136
C06606=1023.546,410.282,345.561,173.745,49.501,160.139
C06607=1023.557,410.528,345.515,173.759,49.503,160.141
C06608=1023.572,410.850,345.455,173.775,49.506,160.145
C06609=1023.585,411.172,345.393,173.791,49.508,160.148
C06610=1023.600,411.493,345.333,173.808,49.511,160.151
C06611=1023.614,411.816,345.271,173.824,49.514,160.155
C06612=1023.625,412.061,345.225,173.836,49.516,160.157
C06613=1023.635,412.306,345.179,173.850,49.518,160.160
C06614=1023.646,412.552,345.131,173.862,49.520,160.163
C06615=1023.657,412.797,345.084,173.874,49.522,160.165
C06616=1023.668,413.042,345.038,173.888,49.524,160.168
C06617=1023.679,413.288,344.991,173.900,49.527,160.171
C06618=1023.690,413.533,344.944,173.913,49.529,160.173
C06619=1023.700,413.778,344.897,173.926,49.531,160.176
C06620=1023.712,414.024,344.850,173.939,49.533,160.179
C06621=1023.723,414.269,344.803,173.952,49.535,160.181
C06622=1023.734,414.514,344.756,173.964,49.537,160.184
C06623=1023.745,414.759,344.710,173.978,49.540,160.187
C06624=1023.756,415.005,344.662,173.991,49.542,160.189
C06625=1023.768,415.251,344.615,174.004,49.544,160.192
C06626=1023.779,415.496,344.569,174.017,49.547,160.195
C06627=1023.790,415.741,344.520,174.030,49.549,160.198
C06628=1023.801,415.987,344.473,174.044,49.551,160.200
C06629=1023.812,416.231,344.426,174.057,49.554,160.203
C06630=1023.823,416.477,344.378,174.070,49.556,160.206
C06631=1023.835,416.722,344.331,174.084,49.558,160.209
C06632=1023.846,416.967,344.283,174.097,49.561,160.212
C06633=1023.857,417.213,344.236,174.110,49.563,160.215
C06634=1023.868,417.458,344.188,174.124,49.566,160.217
C06635=1023.879,417.702,344.140,174.137,49.568,160.220
C06636=1023.891,417.948,344.092,174.151,49.571,160.223
C06637=1023.902,418.193,344.045,174.164,49.573,160.226
C06638=1023.913,418.439,343.997,174.178,49.575,160.229
C06639=1023.925,418.684,343.949,174.192,49.578,160.232
C06640=1023.936,418.929,343.901,174.205,49.581,160.235
C06641=1023.948,419.174,343.853,174.218,49.583,160.238
C06642=1023.959,419.420,343.805,174.233,49.586,160.241
C06643=1023.971,419.664,343.756,174.246,49.588,160.244
C06644=1023.983,419.909,343.708,174.260,49.591,160.247
C06645=1023.994,420.155,343.660,174.274,49.593,160.249
C06646=1024.006,420.400,343.612,174.288,49.596,160.253
C06647=1024.017,420.644,343.563,174.302,49.599,160.255
C06648=1024.029,420.889,343.516,174.316,49.601,160.259
C06649=1024.040,421.135,343.467,174.330,49.604,160.262
C06650=1024.052,421.379,343.419,174.344,49.607,160.265
C06651=1024.064,421.625,343.370,174.358,49.609,160.268
C06652=1024.076,421.870,343.322,174.372,49.612,160.271
C06653=1024.087,422.115,343.274,174.387,49.615,160.274
C06654=1024.099,422.360,343.225,174.401,49.618,160.277
C06655=1024.111,422.604,343.176,174.415,49.620,160.280
C06656=1024.123,422.850,343.127,174.429,49.623,160.283
C06657=1024.134,423.094,343.078,174.444,49.627,160.286
C06658=1024.147,423.339,343.029,174.459,49.629,160.290
C06659=1024.159,423.584,342.980,174.473,49.632,160.293
C06660=1024.170,423.829,342.931,174.487,49.635,160.296
C06661=1024.183,424.074,342.882,174.503,49.638,160.299
C06662=1024.194,424.319,342.833,174.517,49.640,160.302
C06663=1024.206,424.564,342.784,174.531,49.643,160.305
C06664=1024.218,424.809,342.735,174.546,49.646,160.309
C06665=1024.230,425.054,342.686,174.561,49.650,160.312
C06666=1024.242,425.298,342.636,174.576,49.652,160.315
C06667=1024.255,425.543,342.588,174.590,49.655,160.318
C06668=1024.271,425.877,342.520,174.611,49.659,160.323
C06669=1024.287,426.211,342.452,174.631,49.663,160.327
C06670=1024.304,426.543,342.385,174.651,49.668,160.332
C06671=1024.320,426.876,342.317,174.672,49.671,160.336
C06672=1024.333,427.121,342.267,174.687,49.675,160.340
C06673=1024.345,427.366,342.217,174.702,49.678,160.343
C06674=1024.357,427.610,342.168,174.718,49.681,160.347
C06675=1024.369,427.856,342.118,174.733,49.684,160.350
C06676=1024.381,428.100,342.068,174.748,49.688,160.353
C06677=1024.393,428.345,342.018,174.763,49.690,160.357
C06678=1024.406,428.589,341.967,174.779,49.694,160.360
C06679=1024.418,428.834,341.917,174.795,49.697,160.364
C06680=1024.431,429.079,341.868,174.811,49.700,160.367
C06681=1024.444,429.324,341.817,174.826,49.703,160.371
C06682=1024.456,429.568,341.767,174.841,49.707,160.374
C06683=1024.468,429.813,341.717,174.856,49.710,160.378
C06684=1024.481,430.057,341.666,174.872,49.714,160.381
C06685=1024.493,430.302,341.616,174.888,49.717,160.385
C06686=1024.506,430.546,341.566,174.905,49.720,160.389
C06687=1024.518,430.791,341.515,174.920,49.723,160.392
C06688=1024.531,431.036,341.464,174.936,49.726,160.396
C06689=1024.544,431.280,341.413,174.952,49.730,160.399
C06690=1024.557,431.525,341.364,174.968,49.733,160.403
C06691=1024.570,431.769,341.313,174.984,49.737,160.406
C06692=1024.583,432.014,341.262,175.000,49.740,160.410
C06693=1024.595,432.258,341.211,175.017,49.744,160.414
C06694=1024.608,432.502,341.160,175.033,49.747,160.418
C06695=1024.621,432.747,341.109,175.049,49.751,160.421
C06696=1024.634,432.991,341.058,175.066,49.754,160.425
C06697=1024.647,433.236,341.007,175.082,49.758,160.429
C06698=1024.660,433.481,340.956,175.098,49.762,160.432
C06699=1024.673,433.725,340.905,175.115,49.765,160.436
C06700=1024.686,433.969,340.854,175.131,49.769,160.440
C06701=1024.699,434.214,340.803,175.148,49.772,160.444
C06702=1024.712,434.458,340.752,175.164,49.776,160.447
C06703=1024.724,434.703,340.699,175.182,49.779,160.451
C06704=1024.738,434.948,340.648,175.199,49.783,160.455
C06705=1024.751,435.191,340.597,175.215,49.787,160.459
C06706=1024.764,435.435,340.545,175.232,49.790,160.463
C06707=1024.777,435.680,340.493,175.249,49.794,160.467
C06708=1024.791,435.925,340.442,175.266,49.798,160.471
C06709=1024.803,436.169,340.389,175.283,49.801,160.475
C06710=1024.817,436.413,340.338,175.301,49.805,160.479
C06711=1024.830,436.657,340.286,175.318,49.809,160.483
C06712=1024.844,436.901,340.234,175.334,49.813,160.487
C06713=1024.857,437.146,340.182,175.352,49.817,160.491
C06714=1024.871,437.390,340.130,175.369,49.820,160.495
C06715=1024.883,437.635,340.077,175.387,49.824,160.499
C06716=1024.897,437.878,340.025,175.404,49.828,160.503
C06717=1024.911,438.122,339.973,175.422,49.832,160.507
C06718=1024.924,438.367,339.921,175.439,49.836,160.511
C06719=1024.937,438.611,339.868,175.457,49.840,160.515
C06720=1024.951,438.855,339.816,175.475,49.844,160.519
C06721=1024.965,439.099,339.763,175.493,49.848,160.523
C06722=1024.979,439.342,339.711,175.511,49.852,160.527
C06723=1024.992,439.588,339.658,175.529,49.856,160.532
C06724=1025.006,439.831,339.605,175.546,49.860,160.536
C06725=1025.020,440.075,339.553,175.564,49.864,160.540
C06726=1025.033,440.320,339.499,175.583,49.868,160.544
C06727=1025.047,440.563,339.447,175.601,49.872,160.548
C06728=1025.066,440.903,339.373,175.626,49.878,160.554
C06729=1025.086,441.242,339.300,175.652,49.883,160.560
C06730=1025.105,441.581,339.226,175.677,49.889,160.566
C06731=1025.125,441.920,339.152,175.703,49.894,160.572
C06732=1025.139,442.163,339.099,175.721,49.899,160.577
C06733=1025.153,442.406,339.046,175.740,49.902,160.581
C06734=1025.168,442.650,338.993,175.759,49.907,160.585
C06735=1025.182,442.894,338.941,175.778,49.911,160.590
C06736=1025.198,443.137,338.888,175.796,49.915,160.594
C06737=1025.214,443.380,338.837,175.816,49.918,160.598
C06738=1025.230,443.624,338.786,175.835,49.922,160.603
C06739=1025.247,443.868,338.735,175.854,49.926,160.607
C06740=1025.264,444.112,338.685,175.872,49.930,160.611
C06741=1025.282,444.355,338.635,175.892,49.934,160.616
C06742=1025.300,444.599,338.585,175.911,49.937,160.620
C06743=1025.319,444.843,338.536,175.931,49.941,160.625
C06744=1025.338,445.087,338.487,175.951,49.944,160.629
C06745=1025.357,445.332,338.439,175.971,49.947,160.633
C06746=1025.378,445.576,338.390,175.990,49.950,160.637
C06747=1025.398,445.820,338.343,176.010,49.953,160.642
C06748=1025.419,446.064,338.295,176.030,49.957,160.646
C06749=1025.439,446.309,338.249,176.049,49.960,160.650
C06750=1025.462,446.553,338.202,176.070,49.963,160.655
C06751=1025.483,446.798,338.156,176.090,49.966,160.659
C06752=1025.507,447.042,338.110,176.110,49.969,160.663
C06753=1025.529,447.287,338.064,176.131,49.972,160.668
C06754=1025.553,447.532,338.020,176.150,49.975,160.672
C06755=1025.577,447.777,337.976,176.171,49.977,160.676
C06756=1025.601,448.021,337.931,176.191,49.980,160.680
C06757=1025.626,448.267,337.887,176.213,49.982,160.685
C06758=1025.651,448.512,337.843,176.234,49.985,160.689
C06759=1025.677,448.757,337.800,176.254,49.988,160.693
C06760=1025.704,449.002,337.757,176.276,49.990,160.698
C06761=1025.730,449.248,337.716,176.296,49.992,160.702
C06762=1025.758,449.492,337.673,176.318,49.994,160.706
C06763=1025.785,449.738,337.632,176.339,49.997,160.710
C06764=1025.813,449.983,337.591,176.360,49.999,160.715
C06765=1025.841,450.228,337.550,176.382,50.001,160.719
C06766=1025.870,450.474,337.510,176.403,50.003,160.723
C06767=1025.900,450.719,337.470,176.425,50.005,160.727
C06768=1025.930,450.964,337.431,176.446,50.007,160.731
C06769=1025.959,451.210,337.391,176.467,50.009,160.736
C06770=1025.991,451.456,337.352,176.490,50.010,160.740
C06771=1026.022,451.701,337.314,176.511,50.012,160.744
C06772=1025.392,448.754,337.472,176.247,50.048,160.711
C06773=1025.367,448.510,337.515,176.227,50.046,160.707
C06774=1025.342,448.264,337.558,176.205,50.044,160.703
C06775=1025.317,448.019,337.602,176.185,50.041,160.698
C06776=1025.293,447.774,337.645,176.164,50.038,160.694
C06777=1025.268,447.530,337.690,176.144,50.036,160.690
C06778=1025.245,447.285,337.736,176.123,50.033,160.685
C06779=1025.222,447.040,337.781,176.103,50.031,160.681
C06780=1025.199,446.796,337.827,176.083,50.028,160.677
C06781=1025.177,446.550,337.873,176.063,50.025,160.673
C06782=1025.155,446.306,337.919,176.043,50.022,160.668
C06783=1025.134,446.061,337.966,176.022,50.019,160.664
C06784=1025.113,445.817,338.013,176.002,50.016,160.660
C06785=1025.092,445.573,338.060,175.983,50.013,160.656
C06786=1025.072,445.329,338.109,175.963,50.010,160.651
C06787=1025.052,445.085,338.157,175.943,50.006,160.647
C06788=1025.033,444.841,338.206,175.924,50.003,160.643
C06789=1025.015,444.596,338.255,175.904,50.000,160.638
C06790=1024.997,444.352,338.305,175.884,49.996,160.634
C06791=1024.980,444.108,338.354,175.865,49.993,160.630
C06792=1024.962,443.865,338.405,175.846,49.990,160.625
C06793=1024.944,443.621,338.455,175.827,49.986,160.621
C06794=1024.929,443.377,338.507,175.808,49.982,160.617
C06795=1024.913,443.134,338.558,175.789,49.978,160.612
C06796=1024.897,442.890,338.610,175.770,49.974,160.608
C06797=1024.881,442.646,338.662,175.751,49.971,160.604
C06798=1024.867,442.403,338.715,175.732,49.967,160.599
C06799=1024.853,442.160,338.767,175.713,49.962,160.595
C06800=1024.839,441.917,338.821,175.696,49.959,160.591
C06801=1024.821,441.607,338.888,175.671,49.954,160.585
C06802=1024.803,441.296,338.956,175.648,49.948,160.580
C06803=1024.785,440.985,339.024,175.624,49.943,160.574
C06804=1024.768,440.674,339.091,175.601,49.938,160.569
C06805=1024.754,440.430,339.143,175.583,49.934,160.564
C06806=1024.740,440.186,339.196,175.565,49.930,160.560
C06807=1024.727,439.942,339.250,175.546,49.926,160.556
C06808=1024.713,439.698,339.302,175.529,49.922,160.552
C06809=1024.698,439.454,339.355,175.511,49.918,160.548
C06810=1024.685,439.210,339.407,175.492,49.915,160.543
C06811=1024.672,438.966,339.460,175.475,49.911,160.539
C06812=1024.658,438.722,339.513,175.457,49.907,160.535
C06813=1024.644,438.478,339.565,175.439,49.903,160.531
C06814=1024.631,438.234,339.617,175.422,49.899,160.527
C06815=1024.618,437.990,339.670,175.404,49.896,160.523
C06816=1024.604,437.745,339.722,175.386,49.892,160.519
C06817=1024.591,437.501,339.774,175.369,49.888,160.515
C06818=1024.577,437.257,339.826,175.351,49.885,160.511
C06819=1024.563,437.013,339.878,175.334,49.881,160.507
C06820=1024.551,436.769,339.931,175.316,49.877,160.503
C06821=1024.537,436.524,339.983,175.300,49.873,160.499
C06822=1024.524,436.280,340.034,175.283,49.870,160.495
C06823=1024.510,436.036,340.086,175.265,49.866,160.491
C06824=1024.497,435.791,340.138,175.248,49.862,160.487
C06825=1024.484,435.547,340.189,175.231,49.859,160.483
C06826=1024.471,435.303,340.242,175.214,49.855,160.479
C06827=1024.458,435.058,340.293,175.197,49.852,160.476
C06828=1024.445,434.814,340.344,175.180,49.848,160.472
C06829=1024.431,434.570,340.396,175.164,49.844,160.468
C06830=1024.418,434.325,340.447,175.147,49.841,160.464
C06831=1024.406,434.081,340.498,175.130,49.838,160.460
C06832=1024.392,433.836,340.550,175.113,49.834,160.456
C06833=1024.379,433.592,340.601,175.097,49.831,160.453
C06834=1024.366,433.347,340.652,175.080,49.827,160.449
C06835=1024.354,433.103,340.703,175.063,49.824,160.445
C06836=1024.341,432.859,340.755,175.048,49.820,160.442
C06837=1024.327,432.615,340.806,175.031,49.816,160.438
C06838=1024.315,432.369,340.856,175.014,49.813,160.434
C06839=1024.302,432.125,340.907,174.998,49.810,160.430
C06840=1024.289,431.880,340.958,174.983,49.807,160.427
C06841=1024.276,431.636,341.009,174.966,49.804,160.423
C06842=1024.264,431.391,341.059,174.950,49.800,160.419
C06843=1024.251,431.147,341.110,174.934,49.797,160.416
C06844=1024.238,430.902,341.161,174.918,49.793,160.412
C06845=1024.226,430.657,341.211,174.902,49.791,160.409
C06846=1024.213,430.413,341.262,174.886,49.787,160.405
C06847=1024.200,430.168,341.311,174.870,49.784,160.402
C06848=1024.187,429.924,341.362,174.854,49.781,160.398
C06849=1024.175,429.679,341.412,174.838,49.777,160.394
C06850=1024.163,429.435,341.462,174.823,49.775,160.391
C06851=1024.150,429.190,341.512,174.807,49.771,160.387
C06852=1024.138,428.946,341.563,174.792,49.768,160.384
C06853=1024.125,428.701,341.613,174.776,49.765,160.381
C06854=1024.113,428.456,341.663,174.760,49.762,160.377
C06855=1024.101,428.211,341.713,174.745,49.759,160.374
C06856=1024.088,427.967,341.763,174.730,49.756,160.370
C06857=1024.075,427.722,341.813,174.715,49.753,160.367
C06858=1024.063,427.477,341.863,174.699,49.750,160.364
C06859=1024.051,427.233,341.913,174.684,49.747,160.360
C06860=1024.039,426.987,341.962,174.669,49.743,160.357
C06861=1024.022,426.652,342.031,174.648,49.740,160.352
C06862=1024.005,426.316,342.099,174.627,49.735,160.348
C06863=1023.990,425.981,342.167,174.607,49.731,160.343
C06864=1023.973,425.645,342.235,174.586,49.727,160.338
C06865=1023.961,425.401,342.284,174.572,49.724,160.335
C06866=1023.949,425.156,342.333,174.556,49.721,160.332
C06867=1023.937,424.910,342.383,174.542,49.719,160.329
C06868=1023.925,424.666,342.431,174.527,49.716,160.325
C06869=1023.912,424.421,342.481,174.513,49.713,160.322
C06870=1023.901,424.176,342.530,174.497,49.711,160.319
C06871=1023.888,423.931,342.579,174.483,49.707,160.316
C06872=1023.877,423.686,342.628,174.468,49.705,160.313
C06873=1023.865,423.442,342.677,174.454,49.702,160.310
C06874=1023.853,423.197,342.726,174.440,49.699,160.307
C06875=1023.841,422.952,342.775,174.425,49.697,160.303
C06876=1023.830,422.706,342.823,174.410,49.694,160.300
C06877=1023.817,422.461,342.872,174.396,49.691,160.297
C06878=1023.806,422.217,342.921,174.382,49.688,160.294
C06879=1023.795,421.972,342.970,174.367,49.686,160.291
C06880=1023.783,421.727,343.018,174.353,49.683,160.288
C06881=1023.771,421.481,343.067,174.339,49.680,160.285
C06882=1023.759,421.236,343.115,174.325,49.678,160.282
C06883=1023.747,420.992,343.164,174.311,49.675,160.279
C06884=1023.736,420.746,343.211,174.297,49.672,160.276
C06885=1023.724,420.500,343.260,174.282,49.670,160.273
C06886=1023.712,420.256,343.308,174.268,49.667,160.270
C06887=1023.701,420.011,343.357,174.254,49.665,160.267
C06888=1023.689,419.766,343.404,174.241,49.663,160.264
C06889=1023.678,419.520,343.453,174.227,49.660,160.261
C06890=1023.666,419.275,343.500,174.213,49.658,160.258
C06891=1023.655,419.030,343.549,174.199,49.655,160.255
C06892=1023.643,418.785,343.596,174.185,49.653,160.252
C06893=1023.632,418.540,343.644,174.172,49.650,160.249
C06894=1023.621,418.295,343.692,174.158,49.648,160.246
C06895=1023.609,418.050,343.740,174.145,49.645,160.243
C06896=1023.598,417.805,343.788,174.131,49.643,160.240
C06897=1023.586,417.560,343.836,174.117,49.641,160.238
C06898=1023.575,417.314,343.883,174.104,49.638,160.235
C06899=1023.564,417.069,343.931,174.091,49.636,160.232
C06900=1023.553,416.824,343.979,174.077,49.633,160.229
C06901=1023.541,416.578,344.026,174.063,49.631,160.226
C06902=1023.531,416.334,344.074,174.050,49.629,160.223
C06903=1023.519,416.088,344.121,174.037,49.627,160.221
C06904=1023.507,415.843,344.169,174.024,49.624,160.218
C06905=1023.497,415.598,344.216,174.010,49.623,160.215
C06906=1023.485,415.352,344.264,173.998,49.620,160.212
C06907=1023.474,415.107,344.311,173.984,49.618,160.210
C06908=1023.464,414.861,344.358,173.971,49.615,160.207
C06909=1023.452,414.616,344.405,173.958,49.614,160.204
C06910=1023.441,414.371,344.451,173.944,49.611,160.201
C06911=1023.430,414.125,344.498,173.932,49.609,160.199
C06912=1023.419,413.880,344.545,173.919,49.607,160.196
C06913=1023.408,413.634,344.593,173.906,49.605,160.194
C06914=1023.397,413.389,344.639,173.893,49.603,160.191
C06915=1023.386,413.144,344.686,173.880,49.601,160.188
C06916=1023.374,412.899,344.733,173.868,49.599,160.185
C06917=1023.364,412.654,344.779,173.855,49.597,160.183
C06918=1023.353,412.408,344.827,173.842,49.595,160.180
C06919=1023.342,412.162,344.873,173.829,49.593,160.178
C06920=1023.331,411.917,344.920,173.817,49.591,160.175
C06921=1023.317,411.593,344.981,173.800,49.588,160.172
C06922=1023.303,411.268,345.043,173.783,49.585,160.168
C06923=1023.289,410.945,345.104,173.767,49.583,160.165
C06924=1023.275,410.620,345.165,173.750,49.580,160.161
C06925=1023.264,410.375,345.212,173.738,49.579,160.159
C06926=1023.253,410.129,345.258,173.725,49.577,160.156
C06927=1023.242,409.884,345.304,173.712,49.575,160.154
C06928=1023.232,409.639,345.350,173.701,49.573,160.151
C06929=1023.222,409.393,345.397,173.688,49.571,160.149
C06930=1023.211,409.147,345.443,173.676,49.569,160.146
C06931=1023.199,408.901,345.488,173.664,49.567,160.144
C06932=1023.189,408.656,345.534,173.651,49.566,160.141
C06933=1023.178,408.410,345.580,173.639,49.564,160.139
C06934=1023.167,408.165,345.626,173.627,49.562,160.136
C06935=1023.157,407.919,345.672,173.615,49.560,160.134
C06936=1023.147,407.674,345.717,173.603,49.559,160.132
C06937=1023.136,407.428,345.763,173.591,49.557,160.129
C06938=1023.126,407.183,345.809,173.579,49.556,160.127
C06939=1023.115,406.937,345.854,173.567,49.554,160.125
C06940=1023.104,406.691,345.900,173.555,49.552,160.122
C06941=1023.094,406.446,345.945,173.542,49.550,160.120
C06942=1023.084,406.200,345.990,173.531,49.549,160.118
C06943=1023.073,405.955,346.036,173.519,49.547,160.115
C06944=1023.062,405.709,346.082,173.507,49.546,160.113
C06945=1023.053,405.464,346.127,173.495,49.544,160.110
C06946=1023.041,405.218,346.172,173.483,49.543,160.108
C06947=1023.031,404.972,346.218,173.471,49.541,160.106
C06948=1023.021,404.727,346.263,173.460,49.539,160.103
C06949=1023.011,404.481,346.308,173.448,49.538,160.101
C06950=1023.001,404.235,346.353,173.437,49.536,160.099
C06951=1022.990,403.990,346.399,173.425,49.535,160.097
C06952=1022.981,403.744,346.444,173.413,49.534,160.094
C06953=1022.969,403.498,346.488,173.402,49.532,160.092
C06954=1022.960,403.253,346.533,173.390,49.531,160.090
C06955=1022.949,403.007,346.579,173.378,49.529,160.088
C06956=1022.939,402.762,346.624,173.367,49.528,160.085
C06957=1022.930,402.516,346.669,173.356,49.526,160.083
C06958=1022.919,402.270,346.714,173.344,49.525,160.081
C06959=1022.910,402.025,346.759,173.332,49.523,160.079
C06960=1022.899,401.779,346.803,173.322,49.522,160.077
C06961=1022.889,401.533,346.848,173.310,49.521,160.074
C06962=1022.879,401.288,346.893,173.299,49.519,160.072
C06963=1022.869,401.042,346.938,173.288,49.517,160.070
C06964=1022.860,400.796,346.982,173.276,49.516,160.068
C06965=1022.849,400.550,347.027,173.265,49.515,160.066
C06966=1022.839,400.305,347.071,173.254,49.514,160.064
C06967=1022.830,400.058,347.116,173.242,49.513,160.061
C06968=1022.819,399.813,347.160,173.232,49.511,160.059
C06969=1022.810,399.568,347.205,173.220,49.510,160.057
C06970=1022.800,399.322,347.249,173.209,49.509,160.055
C06971=1022.790,399.076,347.293,173.198,49.508,160.053
C06972=1022.780,398.830,347.337,173.187,49.506,160.051
C06973=1022.770,398.583,347.381,173.176,49.505,160.049
C06974=1022.760,398.338,347.426,173.166,49.504,160.047
C06975=1022.751,398.092,347.470,173.154,49.503,160.045
C06976=1022.740,397.846,347.513,173.143,49.502,160.043
C06977=1022.731,397.601,347.558,173.133,49.500,160.041
C06978=1022.721,397.355,347.602,173.122,49.500,160.039
C06979=1022.711,397.109,347.646,173.111,49.498,160.037
C06980=1022.701,396.863,347.689,173.100,49.498,160.035
C06981=1022.690,396.562,347.743,173.087,49.496,160.032
C06982=1022.677,396.260,347.797,173.074,49.495,160.030
C06983=1022.665,395.957,347.850,173.061,49.494,160.027
C06984=1022.654,395.656,347.904,173.047,49.493,160.025
C06985=1022.644,395.410,347.948,173.036,49.491,160.023
C06986=1022.634,395.164,347.992,173.026,49.490,160.021
C06987=1022.624,394.918,348.035,173.015,49.490,160.019
C06988=1022.615,394.673,348.078,173.005,49.489,160.017
C06989=1022.605,394.426,348.122,172.994,49.487,160.015
C06990=1022.595,394.181,348.165,172.984,49.487,160.013
C06991=1022.586,393.934,348.209,172.973,49.486,160.011
C06992=1022.577,393.689,348.252,172.962,49.485,160.009
C06993=1022.567,393.443,348.296,172.952,49.484,160.008
C06994=1022.557,393.196,348.339,172.942,49.483,160.006
C06995=1022.549,392.951,348.383,172.931,49.482,160.004
C06996=1022.539,392.704,348.425,172.921,49.481,160.002
C06997=1022.529,392.459,348.469,172.910,49.481,160.000
C06998=1022.519,392.213,348.511,172.900,49.480,159.998
C06999=1022.510,391.966,348.555,172.890,49.479,159.996
C07000=1022.501,391.721,348.598,172.880,49.478,159.994
C07001=1022.491,391.474,348.641,172.869,49.477,159.993
C07002=1022.482,391.229,348.683,172.859,49.477,159.991
C07003=1022.473,390.982,348.726,172.849,49.476,159.989
C07004=1022.463,390.736,348.769,172.839,49.475,159.987
C07005=1022.453,390.490,348.812,172.828,49.475,159.985
C07006=1022.445,390.244,348.855,172.818,49.474,159.983
C07007=1022.435,389.998,348.898,172.808,49.474,159.982
C07008=1022.426,389.752,348.941,172.798,49.473,159.980
C07009=1022.416,389.506,348.983,172.787,49.472,159.978
C07010=1022.407,389.260,349.027,172.778,49.471,159.976
C07011=1022.398,389.014,349.069,172.767,49.470,159.974
C07012=1022.388,388.767,349.112,172.758,49.470,159.973
C07013=1022.379,388.521,349.153,172.747,49.469,159.971
C07014=1022.370,388.275,349.196,172.737,49.469,159.969
C07015=1022.360,388.029,349.239,172.729,49.468,159.968
C07016=1022.352,387.783,349.282,172.718,49.467,159.966
C07017=1022.343,387.536,349.323,172.709,49.467,159.964
C07018=1022.333,387.290,349.366,172.699,49.467,159.963
C07019=1022.324,387.044,349.409,172.689,49.466,159.961
C07020=1022.315,386.798,349.450,172.679,49.465,159.959
C07021=1022.305,386.552,349.493,172.669,49.465,159.957
C07022=1022.296,386.305,349.535,172.659,49.465,159.956
C07023=1022.287,386.059,349.577,172.649,49.465,159.954
C07024=1022.278,385.813,349.619,172.639,49.464,159.952
C07025=1022.269,385.567,349.661,172.630,49.463,159.951
C07026=1022.260,385.321,349.703,172.620,49.463,159.949
C07027=1022.251,385.075,349.745,172.610,49.462,159.947
C07028=1022.241,384.827,349.787,172.601,49.463,159.946
C07029=1022.232,384.581,349.829,172.591,49.462,159.944
C07030=1022.223,384.335,349.871,172.581,49.462,159.943
C07031=1022.214,384.089,349.913,172.572,49.461,159.941
C07032=1022.204,383.843,349.954,172.563,49.461,159.939
C07033=1022.195,383.597,349.996,172.553,49.460,159.938
C07034=1022.186,383.350,350.037,172.543,49.460,159.936
C07035=1022.178,383.104,350.079,172.534,49.460,159.935
C07036=1022.169,382.857,350.121,172.525,49.460,159.933
C07037=1022.160,382.611,350.163,172.515,49.459,159.931
C07038=1022.150,382.365,350.204,172.505,49.460,159.930
C07039=1022.141,382.119,350.245,172.496,49.459,159.928
C07040=1022.132,381.872,350.286,172.486,49.459,159.927
C07041=1022.123,381.608,350.331,172.477,49.458,159.925
C07042=1022.113,381.343,350.376,172.467,49.459,159.924
C07043=1022.104,381.078,350.420,172.456,49.459,159.922
C07044=1022.095,380.814,350.464,172.446,49.458,159.920
C07045=1022.086,380.567,350.506,172.437,49.458,159.919
C07046=1022.077,380.320,350.547,172.428,49.458,159.917
C07047=1022.068,380.074,350.589,172.419,49.458,159.916
C07048=1022.059,379.828,350.631,172.410,49.457,159.914
C07049=1022.050,379.582,350.671,172.400,49.458,159.913
C07050=1022.042,379.335,350.712,172.390,49.457,159.911
C07051=1022.033,379.088,350.753,172.382,49.457,159.910
C07052=1022.025,378.843,350.795,172.373,49.457,159.908
C07053=1022.017,378.628,350.830,172.365,49.457,159.907
C07054=1022.009,378.414,350.866,172.357,49.457,159.906
C07055=1022.002,378.200,350.901,172.349,49.457,159.905
C07056=1021.994,377.986,350.937,172.341,49.457,159.903
C07057=1021.987,377.772,350.973,172.333,49.456,159.902
C07058=1021.979,377.558,351.008,172.325,49.457,159.901
C07059=1021.972,377.343,351.044,172.318,49.457,159.899
C07060=1021.964,377.130,351.080,172.310,49.457,159.898
C07061=1021.956,376.883,351.121,172.301,49.457,159.897
C07062=1021.948,376.636,351.162,172.292,49.457,159.896
C07063=1021.939,376.390,351.202,172.283,49.457,159.894
C07064=1021.930,376.143,351.243,172.274,49.457,159.893
C07065=1021.921,375.897,351.283,172.265,49.457,159.891
C07066=1021.913,375.650,351.324,172.256,49.457,159.890
C07067=1021.904,375.405,351.364,172.247,49.457,159.889
C07068=1021.895,375.158,351.405,172.238,49.458,159.887
C07069=1021.887,374.912,351.445,172.229,49.457,159.886
C07070=1021.878,374.665,351.486,172.220,49.458,159.884
C07071=1021.869,374.419,351.526,172.212,49.458,159.883
C07072=1021.861,374.171,351.566,172.203,49.458,159.882
C07073=1021.852,373.925,351.606,172.194,49.458,159.880
C07074=1021.843,373.678,351.647,172.186,49.459,159.879
C07075=1021.835,373.432,351.687,172.176,49.459,159.878
C07076=1021.827,373.185,351.727,172.168,49.459,159.876
C07077=1021.818,372.938,351.768,172.160,49.459,159.875
C07078=1021.810,372.692,351.808,172.150,49.460,159.874
C07079=1021.801,372.446,351.848,172.142,49.460,159.873
C07080=1021.793,372.199,351.889,172.134,49.460,159.871
C07081=1021.784,371.952,351.928,172.125,49.461,159.870
C07082=1021.776,371.706,351.969,172.116,49.461,159.869
C07083=1021.768,371.459,352.008,172.108,49.461,159.867
C07084=1021.759,371.212,352.049,172.098,49.462,159.866
C07085=1021.750,370.966,352.088,172.090,49.462,159.865
C07086=1021.742,370.719,352.129,172.082,49.463,159.864
C07087=1021.734,370.473,352.168,172.074,49.462,159.862
C07088=1021.726,370.226,352.208,172.065,49.463,159.861
C07089=1021.717,369.979,352.248,172.056,49.463,159.860
C07090=1021.709,369.732,352.288,172.048,49.464,159.858
C07091=1021.701,369.486,352.328,172.040,49.464,159.857
C07092=1021.693,369.239,352.368,172.031,49.465,159.856
C07093=1021.684,368.993,352.408,172.022,49.465,159.855
C07094=1021.677,368.746,352.448,172.014,49.465,159.854
C07095=1021.668,368.499,352.487,172.006,49.466,159.852
C07096=1021.660,368.252,352.527,171.998,49.466,159.851
C07097=1021.652,368.006,352.566,171.989,49.467,159.850
C07098=1021.643,367.759,352.605,171.981,49.468,159.849
C07099=1021.636,367.512,352.645,171.973,49.468,159.848
C07100=1021.627,367.266,352.685,171.965,49.469,159.846
C07101=1021.616,366.957,352.734,171.954,49.469,159.845
C07102=1021.606,366.650,352.783,171.944,49.470,159.843
C07103=1021.596,366.342,352.832,171.933,49.471,159.842
C07104=1021.585,366.035,352.881,171.923,49.471,159.841
C07105=1021.577,365.788,352.920,171.915,49.472,159.839
C07106=1021.569,365.541,352.959,171.907,49.473,159.838
C07107=1021.561,365.295,352.998,171.899,49.473,159.837
C07108=1021.553,365.048,353.038,171.890,49.474,159.836
C07109=1021.545,364.801,353.076,171.882,49.475,159.835
C07110=1021.536,364.555,353.115,171.874,49.476,159.834
C07111=1021.528,364.308,353.155,171.866,49.476,159.833
C07112=1021.520,364.061,353.193,171.858,49.477,159.832
C07113=1021.512,363.814,353.233,171.850,49.478,159.831
C07114=1021.504,363.567,353.272,171.842,49.478,159.829
C07115=1021.496,363.321,353.311,171.834,49.479,159.828
C07116=1021.488,363.074,353.350,171.826,49.480,159.827
C07117=1021.480,362.826,353.388,171.818,49.480,159.826
C07118=1021.472,362.580,353.427,171.810,49.481,159.825
C07119=1021.464,362.333,353.466,171.802,49.482,159.824
C07120=1021.456,362.086,353.506,171.794,49.482,159.823
C07121=1021.448,361.839,353.544,171.786,49.483,159.822
C07122=1021.440,361.593,353.582,171.778,49.484,159.821
C07123=1021.432,361.346,353.622,171.770,49.485,159.820
C07124=1021.424,361.099,353.660,171.763,49.486,159.819
C07125=1021.416,360.852,353.699,171.754,49.487,159.818
C07126=1021.408,360.605,353.737,171.747,49.488,159.817
C07127=1021.401,360.358,353.776,171.739,49.488,159.816
C07128=1021.393,360.112,353.815,171.731,49.489,159.815
C07129=1021.385,359.864,353.854,171.723,49.490,159.814
C07130=1021.377,359.618,353.892,171.715,49.491,159.813
C07131=1021.369,359.371,353.931,171.707,49.492,159.812
C07132=1021.361,359.124,353.969,171.699,49.493,159.811
C07133=1021.353,358.877,354.008,171.692,49.494,159.810
C07134=1021.345,358.629,354.045,171.684,49.495,159.809
C07135=1021.337,358.383,354.083,171.676,49.496,159.808
C07136=1021.329,358.136,354.122,171.668,49.497,159.807
C07137=1021.321,357.889,354.160,171.660,49.498,159.806
C07138=1021.313,357.642,354.199,171.653,49.499,159.805
C07139=1021.306,357.395,354.237,171.645,49.500,159.804
C07140=1021.298,357.148,354.275,171.637,49.501,159.803
C07141=1021.289,356.901,354.313,171.629,49.502,159.802
C07142=1021.282,356.655,354.351,171.622,49.503,159.801
C07143=1021.274,356.407,354.389,171.615,49.504,159.800
C07144=1021.267,356.161,354.427,171.607,49.506,159.799
C07145=1021.258,355.913,354.465,171.600,49.507,159.798
C07146=1021.251,355.666,354.503,171.592,49.508,159.797
C07147=1021.242,355.419,354.541,171.584,49.509,159.796
C07148=1021.235,355.172,354.579,171.576,49.510,159.795
C07149=1021.227,354.926,354.617,171.569,49.511,159.794
C07150=1021.220,354.678,354.655,171.561,49.512,159.793
C07151=1021.212,354.431,354.693,171.555,49.513,159.793
C07152=1021.204,354.184,354.730,171.547,49.515,159.792
C07153=1021.196,353.938,354.768,171.539,49.516,159.791
C07154=1021.189,353.690,354.806,171.531,49.517,159.790
C07155=1021.181,353.443,354.843,171.524,49.518,159.789
C07156=1021.173,353.196,354.880,171.516,49.519,159.788
C07157=1021.165,352.955,354.918,171.510,49.521,159.787
C07158=1021.158,352.714,354.955,171.502,49.522,159.786
C07159=1021.150,352.473,354.991,171.494,49.523,159.785
C07160=1021.143,352.231,355.028,171.488,49.524,159.785
C07161=1021.135,351.990,355.064,171.480,49.525,159.784
C07162=1021.128,351.749,355.100,171.473,49.527,159.783
C07163=1021.121,351.507,355.137,171.466,49.529,159.782
C07164=1021.113,351.266,355.173,171.459,49.530,159.781
C07165=1021.105,351.019,355.212,171.451,49.531,159.781
C07166=1021.097,350.772,355.249,171.444,49.532,159.780
C07167=1021.090,350.525,355.286,171.437,49.534,159.779
C07168=1021.083,350.278,355.324,171.429,49.535,159.778
C07169=1021.075,350.031,355.361,171.422,49.536,159.777
C07170=1021.067,349.784,355.398,171.416,49.538,159.777
C07171=1021.060,349.537,355.435,171.408,49.539,159.776
C07172=1021.052,349.289,355.472,171.400,49.541,159.775
C07173=1021.045,349.042,355.510,171.393,49.542,159.774
C07174=1021.037,348.795,355.546,171.386,49.543,159.773
C07175=1021.030,348.548,355.584,171.379,49.545,159.772
C07176=1021.022,348.302,355.621,171.371,49.546,159.772
C07177=1021.015,348.054,355.658,171.364,49.548,159.771
C07178=1021.008,347.807,355.695,171.357,49.549,159.770
C07179=1021.000,347.560,355.732,171.350,49.551,159.769
C07180=1020.993,347.313,355.770,171.343,49.552,159.768
C07181=1020.985,347.065,355.806,171.336,49.554,159.768
C07182=1020.977,346.818,355.843,171.329,49.555,159.767
C07183=1020.970,346.571,355.880,171.321,49.557,159.766
C07184=1020.962,346.324,355.917,171.314,49.559,159.765
C07185=1020.954,346.076,355.953,171.308,49.560,159.765
C07186=1020.947,345.829,355.990,171.300,49.562,159.764
C07187=1020.939,345.582,356.027,171.293,49.564,159.763
C07188=1020.931,345.335,356.064,171.286,49.565,159.763
C07189=1020.925,345.087,356.100,171.279,49.567,159.762
C07190=1020.917,344.840,356.137,171.272,49.568,159.761
C07191=1020.910,344.593,356.174,171.265,49.570,159.760
C07192=1020.903,344.346,356.210,171.258,49.571,159.760
C07193=1020.895,344.099,356.247,171.250,49.573,159.759
C07194=1020.888,343.851,356.284,171.244,49.574,159.758
C07195=1020.880,343.604,356.320,171.237,49.577,159.758
C07196=1020.873,343.358,356.356,171.230,49.578,159.757
C07197=1020.866,343.110,356.393,171.223,49.580,159.756
C07198=1020.858,342.863,356.429,171.216,49.581,159.755
C07199=1020.850,342.615,356.466,171.208,49.583,159.755
C07200=1020.843,342.368,356.502,171.202,49.585,159.754
C07201=1020.836,342.121,356.539,171.195,49.587,159.753
C07202=1020.828,341.874,356.575,171.189,49.588,159.753
C07203=1020.821,341.626,356.612,171.182,49.591,159.752
C07204=1020.814,341.379,356.648,171.174,49.592,159.751
C07205=1020.807,341.132,356.684,171.168,49.594,159.751
C07206=1020.799,340.884,356.720,171.161,49.596,159.750
C07207=1020.792,340.638,356.756,171.154,49.597,159.749
C07208=1020.785,340.390,356.793,171.147,49.600,159.749
C07209=1020.778,340.143,356.829,171.140,49.601,159.748
C07210=1020.770,339.896,356.865,171.134,49.603,159.747
C07211=1020.762,339.648,356.901,171.127,49.605,159.747
C07212=1020.755,339.402,356.937,171.120,49.606,159.746
C07213=1020.749,339.153,356.973,171.113,49.609,159.745
C07214=1020.742,338.906,357.009,171.106,49.611,159.745
C07215=1020.734,338.659,357.045,171.100,49.612,159.744
C07216=1020.726,338.411,357.082,171.093,49.615,159.744
C07217=1020.719,338.169,357.117,171.086,49.616,159.743
C07218=1020.712,337.926,357.152,171.079,49.618,159.742
C07219=1020.705,337.684,357.186,171.073,49.620,159.742
C07220=1020.698,337.441,357.222,171.066,49.622,159.741
C07221=1020.691,337.198,357.257,171.060,49.624,159.741
C07222=1020.683,336.956,357.292,171.054,49.626,159.740
C07223=1020.676,336.713,357.327,171.047,49.628,159.740
C07224=1020.669,336.470,357.362,171.040,49.630,159.739
C07225=1020.662,336.222,357.398,171.033,49.632,159.738
C07226=1020.655,335.975,357.434,171.027,49.634,159.738
C07227=1020.648,335.727,357.469,171.020,49.636,159.737
C07228=1020.641,335.480,357.505,171.014,49.638,159.737
C07229=1020.634,335.233,357.540,171.007,49.641,159.736
C07230=1020.626,334.985,357.576,171.001,49.642,159.736
C07231=1020.619,334.738,357.612,170.994,49.644,159.735
C07232=1020.612,334.490,357.647,170.988,49.646,159.734
C07233=1020.605,334.243,357.683,170.981,49.649,159.734
C07234=1020.598,333.996,357.718,170.975,49.651,159.733
C07235=1020.591,333.748,357.754,170.968,49.653,159.733
C07236=1020.584,333.501,357.789,170.962,49.655,159.732
C07237=1020.577,333.254,357.824,170.955,49.657,159.732
C07238=1020.570,333.006,357.860,170.949,49.659,159.731
C07239=1020.562,332.759,357.895,170.942,49.662,159.731
C07240=1020.555,332.512,357.930,170.936,49.664,159.730
C07241=1020.548,332.264,357.966,170.929,49.666,159.730
C07242=1020.541,332.016,358.001,170.923,49.668,159.729
C07243=1020.533,331.769,358.036,170.916,49.670,159.729
C07244=1020.527,331.522,358.071,170.910,49.673,159.728
C07245=1020.520,331.275,358.106,170.903,49.675,159.728
C07246=1020.512,331.027,358.141,170.897,49.677,159.727
C07247=1020.505,330.780,358.176,170.890,49.680,159.727
C07248=1020.498,330.532,358.211,170.884,49.681,159.726
C07249=1020.491,330.285,358.246,170.877,49.684,159.726
C07250=1020.484,330.037,358.282,170.871,49.686,159.725
C07251=1020.476,329.790,358.316,170.864,49.689,159.725
C07252=1020.470,329.542,358.351,170.858,49.691,159.724
C07253=1020.463,329.295,358.386,170.851,49.694,159.724
C07254=1020.455,329.048,358.421,170.845,49.696,159.723
C07255=1020.449,328.800,358.455,170.838,49.698,159.723
C07256=1020.442,328.553,358.491,170.833,49.701,159.723
C07257=1020.435,328.305,358.526,170.826,49.703,159.722
C07258=1020.427,328.057,358.561,170.820,49.706,159.722
C07259=1020.421,327.810,358.596,170.814,49.708,159.721
C07260=1020.414,327.562,358.630,170.807,49.710,159.721
C07261=1020.407,327.315,358.665,170.801,49.713,159.720
C07262=1020.400,327.068,358.700,170.794,49.715,159.720
C07263=1020.393,326.820,358.735,170.789,49.718,159.719
C07264=1020.387,326.572,358.769,170.782,49.720,159.719
C07265=1020.379,326.325,358.804,170.776,49.723,159.719
C07266=1020.372,326.078,358.838,170.769,49.725,159.718
C07267=1020.365,325.830,358.873,170.763,49.727,159.718
C07268=1020.358,325.583,358.907,170.758,49.730,159.717
C07269=1020.351,325.335,358.941,170.751,49.733,159.717
C07270=1020.343,325.088,358.975,170.745,49.735,159.717
C07271=1020.337,324.840,359.009,170.738,49.738,159.716
C07272=1020.329,324.593,359.044,170.733,49.741,159.716
C07273=1020.322,324.345,359.078,170.726,49.744,159.715
C07274=1020.316,324.097,359.112,170.720,49.746,159.715
C07275=1020.308,323.850,359.147,170.713,49.749,159.715
C07276=1020.301,323.602,359.181,170.708,49.751,159.714
C07277=1020.294,323.357,359.214,170.701,49.754,159.714
C07278=1020.287,323.112,359.248,170.695,49.757,159.714
C07279=1020.280,322.867,359.282,170.689,49.759,159.713
C07280=1020.273,322.622,359.315,170.683,49.762,159.713
C07281=1020.266,322.377,359.350,170.677,49.764,159.712
C07282=1020.259,322.132,359.383,170.671,49.767,159.712
C07283=1020.252,321.888,359.417,170.665,49.770,159.712
C07284=1020.246,321.642,359.451,170.659,49.773,159.712
C07285=1020.239,321.395,359.484,170.653,49.775,159.711
C07286=1020.232,321.147,359.518,170.647,49.778,159.711
C07287=1020.224,320.899,359.552,170.641,49.781,159.711
C07288=1020.218,320.651,359.586,170.634,49.784,159.710
C07289=1020.211,320.405,359.621,170.629,49.787,159.710
C07290=1020.204,320.157,359.654,170.623,49.789,159.710
C07291=1020.197,319.909,359.689,170.616,49.792,159.709
C07292=1020.190,319.661,359.723,170.611,49.795,159.709
C07293=1020.184,319.415,359.756,170.604,49.798,159.709
